(* Logix 5000 project; controller CLASE_1 Emulate 5570 rev 28.11; software revision 28.02; part 5 of 15 *)
(* tags used below, declared in another part *)
   P_Intlk : BOOL;   // Unique Parameter Name for auto - discovery
(* P_Intlk, continued *)

ROUTINE Prescan   (* ladder *)
// Clear "lurking" Commands
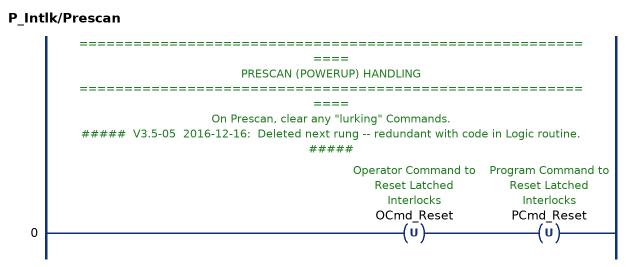
   // ============================================================
   // PRESCAN (POWERUP) HANDLING
   // ============================================================
   // On Prescan, clear any "lurking" Commands.
   // #####  V3.5-05  2016-12-16:  Deleted next rung -- redundant with code in Logic routine.  #####
   0: OTU(OCmd_Reset)OTU(PCmd_Reset);
END_ROUTINE
END_ADD_ON_INSTRUCTION

ADD_ON_INSTRUCTION P_Mode   (* revision 3.5 01 Release, vendor Rockwell Automation, ExecutePrescan, ExecuteEnableInFalse *)
// Mode
// Revision note:
// See V3.5-xx Release Notes for details. Unmodified, up-rev only for V3.5-01 Release.
// Help:
// Copyright © Rockwell Automation, Inc.  All Rights Reserved.
// This instruction provides selection of Mode (owner) for a Device level
// object  (from highest priority to lowest):
// *  No Mode (no owner, EnableIn is false)
// *  Hand (typically tracks hardwired control of device)
// *  Maint (Maintenance) (taken out of normal service for maintenance)
// *  Ovrd (Override) (typically used for process overrides)
// *  Prog  (Program) (automated control, and default if Cfg_ProgNorm = 1)
// *  Oper (Operator (manual control, and default if Cfg_ProgNorm = 0)
// (Program and Operator have the same priority.)
// The current mode is shown with Status bits and also as the primary
// Value for the instruction: an enumeration "Val" as follows:
//   0 = No Mode,
//   1 = Hand,
//   2 = Maintenance,
//   3 = Override,
//   4 = Program (Locked),
//   5 = Operator (Locked),
//   6 = Program (Unlocked, Oper default),
//   7 = Operator (Unlocked, Prog default),
//   8 = Program (Unlocked, = default),
//   9 = Operator (Unlocked, = default).
// When EnableIn is false, all ownership acquire/release and lock/unlock
// Commands are processed "behind the scenes", but the Mode is shown
// as "No Mode" (no owner).  When EnableIn becomes true, the Mode
// takes into account the Commands received -- in other words, the Mode
// becomes the one that would have been in effect had the EnableIn
// False / No Mode condition never occurred.
VAR_INPUT
   Inp_Hand : BOOL; {visible}   // 1=Acquire Hand (typ. hardwired local) Mode, 0=Release Hand Mode
   Inp_Ovrd : BOOL; {visible}   // 1=Acquire Override (higher priority program logic) Mode, 0=Release Override Mode
   Cfg_PCmdClear : BOOL := 1;   // 1=Clear Program Command on receipt; 0=Use Level-based (maintained) PCmds
   Cfg_OvrdOverLock : BOOL := 1;   // 1=Override supersedes Prog/Oper Lock, 0=don't override Lock
   Cfg_ProgDefault : BOOL;   // Default Mode: 1=Program Mode if no requests; 0=Operator Mode if no requests
   PCmd_Acq : BOOL;   // Program Command to Acquire Ownership (Oper to Prog)
   PCmd_Rel : BOOL;   // Program Command to Release Ownership (Prog to Oper)
   PCmd_Lock : BOOL;   // Program Command to Lock Mode in Prog
   PCmd_Unlock : BOOL;   // Program Command to Unlock Mode
   MCmd_Acq : BOOL;   // Maintenance Command to Acquire Ownership (Oper/Prog/Ovrd to Maint)
   MCmd_Rel : BOOL;   // Maintenance Command to Release Ownership (Maint to Oper/Prog/Ovrd)
   OCmd_AcqLock : BOOL;   // Operator Command to Acquire (Prog to Oper) / Lock Ownership
   OCmd_UnlockRel : BOOL;   // Operator Command to Unlock / Release (Oper to Prog) Ownership
END_VAR
VAR_OUTPUT
   Val : SINT; {access Read Only}   // Mode enum: 0=No, 1=H, 2=M, 3=!, 4=P Lock, 5=O Lock, 6=P (O Def), 7=O (P Def), 8=P (= Def), 9=O (= Def)
   Sts_Hand : BOOL; {access Read Only, visible}   // 1=Mode is Hand (supersedes Maint, Ovrd, Prog, Oper)
   Sts_Maint : BOOL; {access Read Only, visible}   // 1=Mode is Maintenance (supersedes Ovrd, Prog, Oper)
   Sts_Ovrd : BOOL; {access Read Only, visible}   // 1=Mode is Override (supersedes Prog, Oper)
   Sts_Prog : BOOL; {access Read Only, visible}   // 1=Mode is Program
   Sts_Oper : BOOL := 1; {access Read Only, visible}   // 1=Mode is Operator
   Sts_ProgOperLock : BOOL; {access Read Only, visible}   // 1=Program or Operator has requested Mode Lock
   Sts_ProgOperSel : BOOL; {access Read Only}   // Prog/Oper selection 1=Program, 0=Operator
   Sts_NoMode : BOOL; {access Read Only}   // 1=Mode is No Mode (no owner, disabled or not scanned)
   Sts_MAcqRcvd : BOOL; {access Read Only}   // 1=Maintenance Acquire command received this scan
   Rdy_MAcq : BOOL; {access Read Only}   // 1=Ready for MCmd_Acq, enable button
   Rdy_MRel : BOOL; {access Read Only}   // 1=Ready for MCmd_Rel, enable button
   Rdy_OAcq : BOOL; {access Read Only}   // 1=Ready for OCmd_AcqLock, enable Acquire (to Oper) button
   Rdy_OLock : BOOL; {access Read Only}   // 1=Ready for OCmd_AcqLock, enable Oper Lock button
   Rdy_OUnlock : BOOL; {access Read Only}   // 1=Ready for OCmd_UnlockRel, enable Oper Unlock button
   Rdy_ORel : BOOL; {access Read Only}   // 1=Ready for OCmd_UnlockRel, enable Release (to Prog) button
   P_Mode : BOOL;   // Unique Parameter Name for auto - discovery
END_VAR
VAR
   Wrk_Locked : BOOL; {access None}   // 1=Program/Operator Mode selection is Locked
   Wrk_Prog : BOOL; {access None}   // Internal Program (1) / Operator (0) Mode selection
   Wrk_Maint : BOOL; {access None}   // Internal Maintenance Mode
   Inf_Lib : STRING_12 := 'RA-BAS'; {access Read Only}   // Display Library for Faceplate call-up
   Inf_Type : STRING_16 := 'P_Mode'; {access Read Only}   // Must contain AOI name, used for HMI and Information S/W
END_VAR

ROUTINE EnableInFalse   (* ladder *)
// Processes received Commands, but shows "NO mode" (no owner)
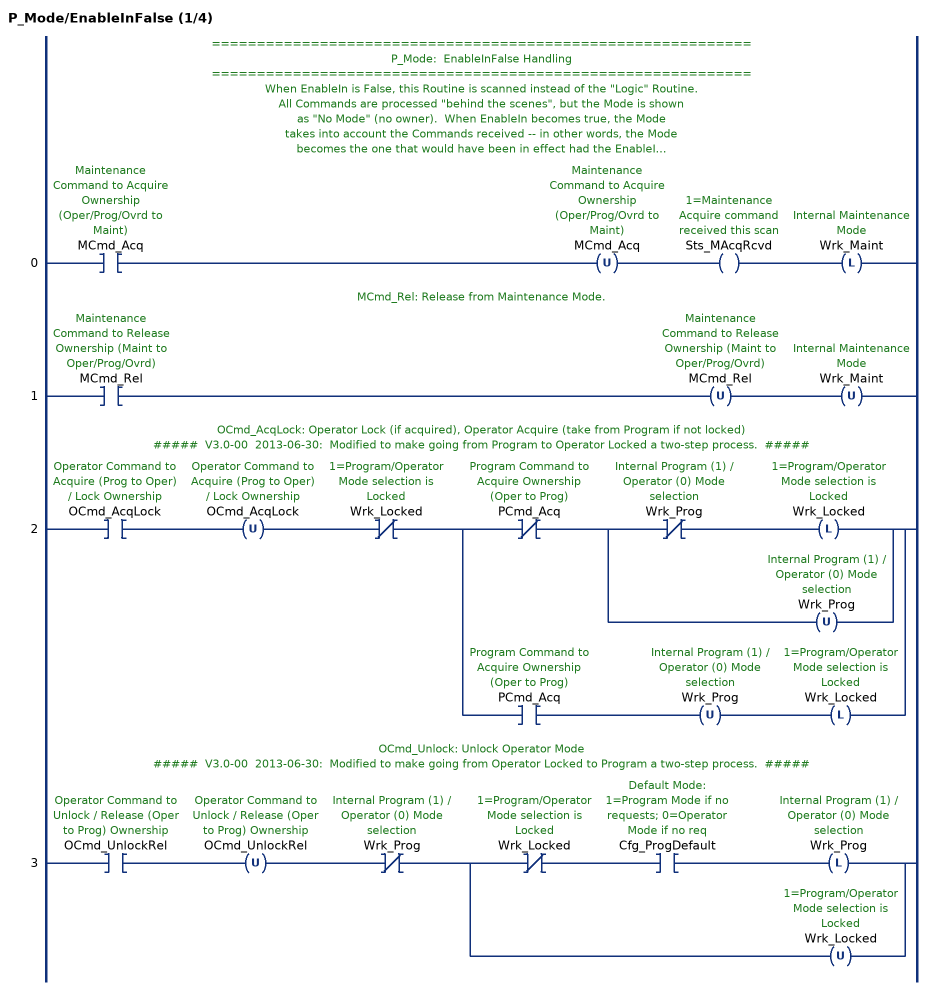
   // ============================================================
   // P_Mode:  EnableInFalse Handling
   // ============================================================
   // When EnableIn is False, this Routine is scanned instead of the "Logic" Routine.
   // All Commands are processed "behind the scenes", but the Mode is shown
   // as "No Mode" (no owner).  When EnableIn becomes true, the Mode
   // takes into account the Commands received -- in other words, the Mode
   // becomes the one that would have been in effect had the EnableIn
   // False / No Mode condition never occurred.
   // ============================================================
   // COMMAND HANDLING
   // ============================================================
   // NOTE:  These rungs MUST be in the order given to meet the following
   // multiple-actions-at-the-same-time scenarios:
   // * Maintenance Release beats Maintenance Acquire
   // * Program Release beats Program Acquire
   // * Program Unlock beats Program Lock
   // * Operator Unlock beats Operator Acquire and Lock (results in Oper Unlocked)
   // * Operator Acquire/Lock must come after Program Unlock
   // * Program Acquire must come after Operator Unlock
   // ===========================================================
   // MCmd_Acq: Acquire for Maintenance Mode, and blink the status
   // that indicates a Maintenance Acquire command was received.
   // #####  V3.1-00  2014-06-30:  Added Sts_MAcqRcvd  #####
   0: XIC(MCmd_Acq)OTU(MCmd_Acq)OTE(Sts_MAcqRcvd)OTL(Wrk_Maint);
   // MCmd_Rel: Release from Maintenance Mode.
   1: XIC(MCmd_Rel)OTU(MCmd_Rel)OTU(Wrk_Maint);
   // OCmd_AcqLock: Operator Lock (if acquired), Operator Acquire (take from Program if not locked)
   // #####  V3.0-00  2013-06-30:  Modified to make going from Program to Operator Locked a two-step process.  #####
   2: XIC(OCmd_AcqLock)OTU(OCmd_AcqLock)XIO(Wrk_Locked)[XIO(PCmd_Acq) [XIO(Wrk_Prog) OTL(Wrk_Locked) ,OTU(Wrk_Prog) ] ,XIC(PCmd_Acq) OTU(Wrk_Prog) OTL(Wrk_Locked) ];
   // OCmd_Unlock: Unlock Operator Mode
   // #####  V3.0-00  2013-06-30:  Modified to make going from Operator Locked to Program a two-step process.  #####
   3: XIC(OCmd_UnlockRel)OTU(OCmd_UnlockRel)XIO(Wrk_Prog)[XIO(Wrk_Locked) XIC(Cfg_ProgDefault) OTL(Wrk_Prog) ,OTU(Wrk_Locked) ];
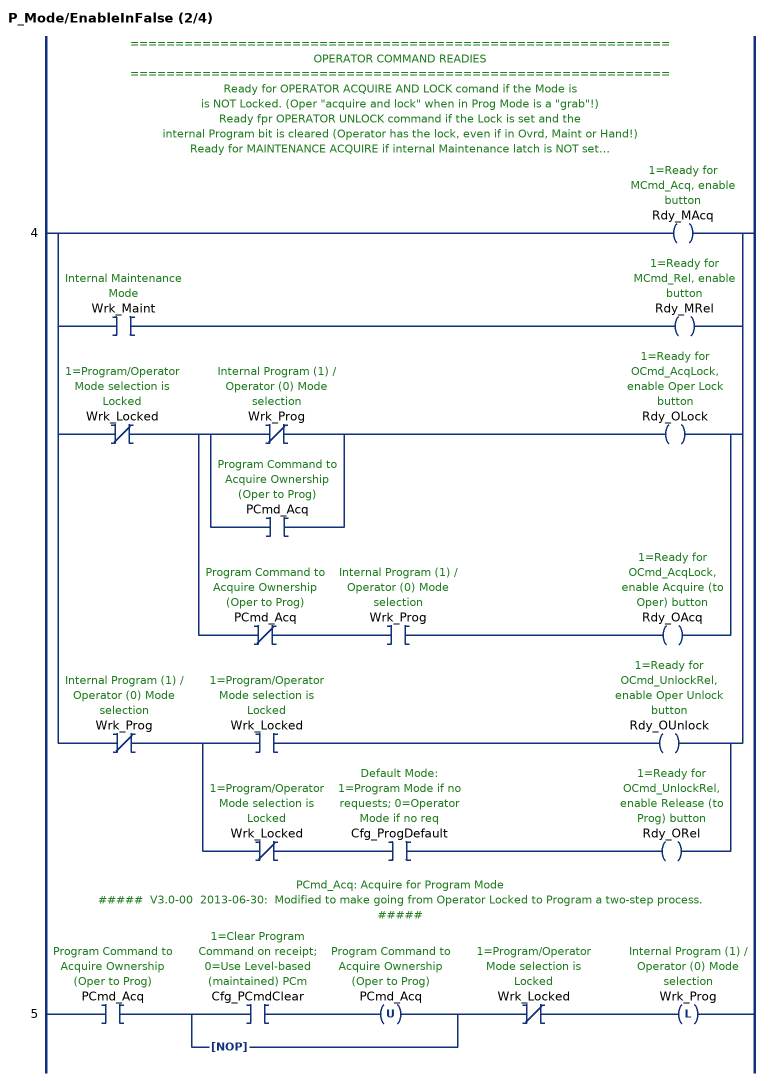
   // ============================================================
   // OPERATOR COMMAND READIES
   // ============================================================
   // Ready for OPERATOR ACQUIRE AND LOCK comand if the Mode is
   //  is NOT Locked. (Oper "acquire and lock" when in Prog Mode is a "grab"!)
   // Ready fpr OPERATOR UNLOCK command if the Lock is set and the
   // internal Program bit is cleared (Operator has the lock, even if in Ovrd, Maint or Hand!)
   // Ready for MAINTENANCE ACQUIRE if internal Maintenance latch is NOT set.
   // But we need to display Ready even if latch IS set so that Sts_MAcqRcvd
   // can blink to reset an external Maintenance expiration timer!!!
   // Ready for MAINTENANCE RELEASE if internal Maintenance latch IS set.
   // #####  V3.0-00  2013-06-30:  Modified Rdy_Unlock for two-step Operator Locked to Program process.  #####
   // #####  V3.1-00  2014-06-30:  Added Sts_MAcqRcvd  #####
   4: [OTE(Rdy_MAcq) ,XIC(Wrk_Maint) OTE(Rdy_MRel) ,XIO(Wrk_Locked) [[XIO(Wrk_Prog) ,XIC(PCmd_Acq) ] OTE(Rdy_OLock) ,XIO(PCmd_Acq) XIC(Wrk_Prog) OTE(Rdy_OAcq) ] ,XIO(Wrk_Prog) [XIC(Wrk_Locked) OTE(Rdy_OUnlock) ,XIO(Wrk_Locked) XIC(Cfg_ProgDefault) OTE(Rdy_ORel) ] ];
   // PCmd_Acq: Acquire for Program Mode
   // #####  V3.0-00  2013-06-30:  Modified to make going from Operator Locked to Program a two-step process.  #####
   5: XIC(PCmd_Acq)[XIC(Cfg_PCmdClear) OTU(PCmd_Acq) ,NOP() ]XIO(Wrk_Locked)OTL(Wrk_Prog);
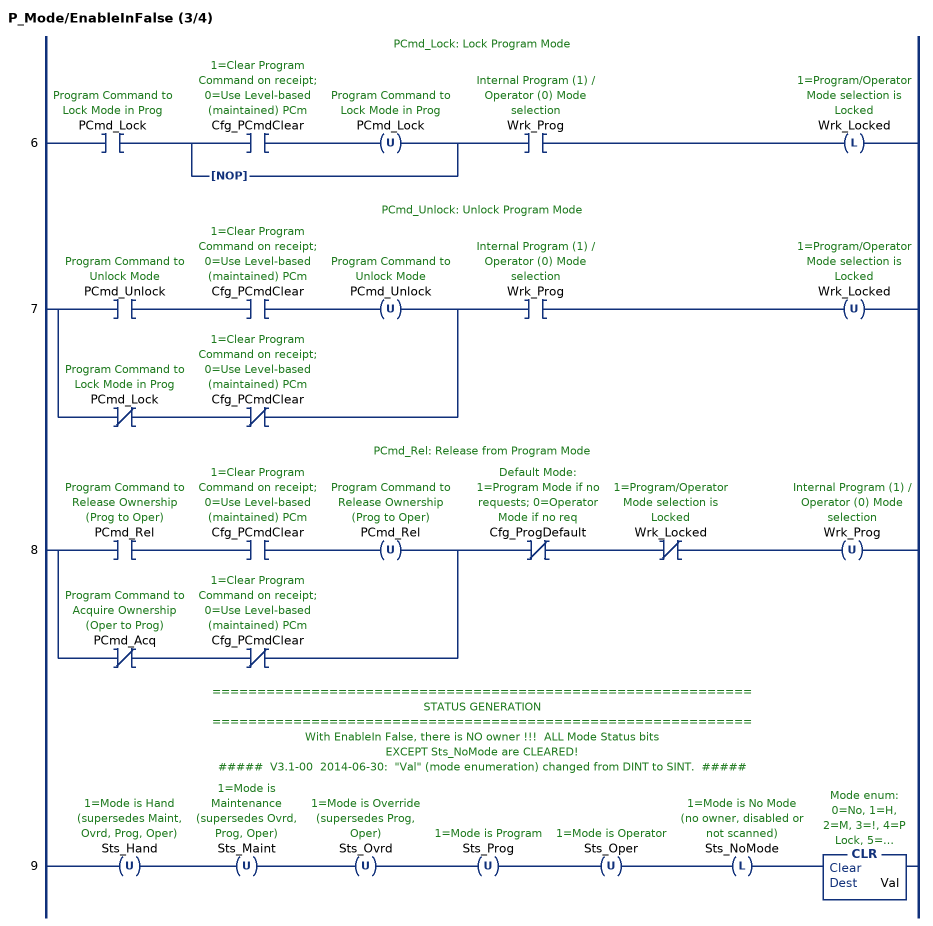
   // PCmd_Lock: Lock Program Mode
   6: XIC(PCmd_Lock)[XIC(Cfg_PCmdClear) OTU(PCmd_Lock) ,NOP() ]XIC(Wrk_Prog)OTL(Wrk_Locked);
   // PCmd_Unlock: Unlock Program Mode
   7: [XIC(PCmd_Unlock) XIC(Cfg_PCmdClear) OTU(PCmd_Unlock) ,XIO(PCmd_Lock) XIO(Cfg_PCmdClear) ]XIC(Wrk_Prog)OTU(Wrk_Locked);
   // PCmd_Rel: Release from Program Mode
   8: [XIC(PCmd_Rel) XIC(Cfg_PCmdClear) OTU(PCmd_Rel) ,XIO(PCmd_Acq) XIO(Cfg_PCmdClear) ]XIO(Cfg_ProgDefault)XIO(Wrk_Locked)OTU(Wrk_Prog);
   // ============================================================
   // STATUS GENERATION
   // ============================================================
   // With EnableIn False, there is NO owner !!!  ALL Mode Status bits
   // EXCEPT Sts_NoMode are CLEARED!
   // #####  V3.1-00  2014-06-30:  "Val" (mode enumeration) changed from DINT to SINT.  #####
   9: OTU(Sts_Hand)OTU(Sts_Maint)OTU(Sts_Ovrd)OTU(Sts_Prog)OTU(Sts_Oper)OTL(Sts_NoMode)CLR(Val);
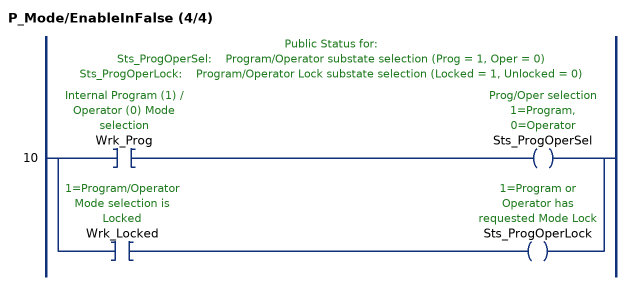
   // Public Status for:
   // Sts_ProgOperSel:    Program/Operator substate selection (Prog = 1, Oper = 0)
   // Sts_ProgOperLock:    Program/Operator Lock substate selection (Locked = 1, Unlocked = 0)
   10: [XIC(Wrk_Prog) OTE(Sts_ProgOperSel) ,XIC(Wrk_Locked) OTE(Sts_ProgOperLock) ];
END_ROUTINE

ROUTINE Logic   (* ladder *)
// Selects Modes (Hand, Maint, Ovrd, Oper, Prog) based on Inputs and Commands
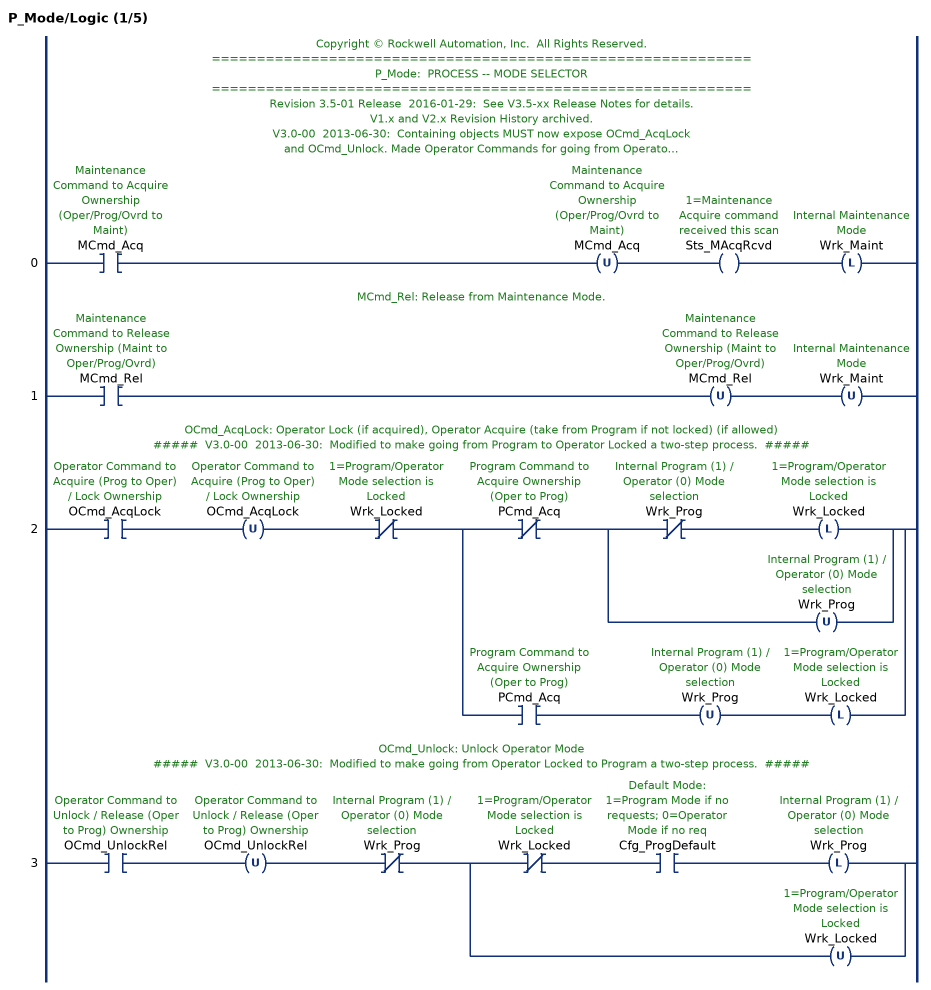
   // Copyright © Rockwell Automation, Inc.  All Rights Reserved.
   // ============================================================
   // P_Mode:  PROCESS -- MODE SELECTOR
   // ============================================================
   // Revision 3.5-01 Release  2016-01-29:  See V3.5-xx Release Notes for details.
   // V1.x and V2.x Revision History archived.
   // V3.0-00  2013-06-30:  Containing objects MUST now expose OCmd_AcqLock
   // and OCmd_Unlock. Made Operator Commands for going from Operator
   // Locked to Program (unlocked) and Program (unlocked) to Operator
   // Lock two-step processes.  Added Inf_Lib, Inf_Type.
   // V3.1-00  2014-06-30:  Containing objects must expose Maintenance Acquire /
   // Release commands and new Sts_MAcqRcvd.
   // Changed Val (enum) to SINT. Fixed parameter descriptions.
   // V3.1-01  2014-09-03:  Unmodified, up-rev only for V3.1-01 public release.
   // V3.5-01  2016-01-29:  Unmodified, up-rev only for V3.5-01 Release.
   // ============================================================
   // This instruction provides selection of Mode (owner) for a Device level
   // object  (from highest priority to lowest):
   // * NO Mode (EnableIn is false)
   // *  Hand (typically tracks hardwired control of device)
   // *  Maint (Maintenance) (taken out of normal service for maintenance)
   // *  Ovrd (Override) (typically used for process overrides)
   // *  Prog  (Program) (automated control, and default if Cfg_ProgNorm = 1)
   // *  Oper (Operator (manual control, and default if Cfg_ProgNorm = 0)
   // The current mode is shown with Status bits and also as the
   // primary Value for the instruction: an enumeration as follows:
   // 0 = No Mode, 1 = Hand, 2 = Maintenance, 3 = Override,
   // 4 = Program (Locked), 5 = Operator (Locked),
   // 6 = Program (Unlocked, Oper default), 7 = Operator (Unlocked, Prog default),
   // 8 = Program (Unlocked, Prog default), 9 = Operator (Unlocked, Oper default).
   // ============================================================
   // COMMAND HANDLING
   // ============================================================
   // NOTE:  These rungs MUST be in the order given to meet the following
   // multiple-actions-at-the-same-time scenarios:
   // * Maintenance Release beats Maintenance Acquire
   // * Program Release beats Program Acquire
   // * Program Unlock beats Program Lock
   // * Operator Unlock beats Operator Acquire / Lock (results in Oper Unlocked)
   // * Program Acquire must come after Operator Unlock
   // If Cfg_ProgDefault = 1, the Mode defaults to Program
   // (instead of Operator) if all other Modes release their requests.
   // ============================================================
   // MCmd_Acq: Acquire for Maintenance Mode, and blink the status
   // that indicates a Maintenance Acquire command was received.
   // #####  V3.1-00  2014-06-30:  Added Sts_MAcqRcvd  #####
   0: XIC(MCmd_Acq)OTU(MCmd_Acq)OTE(Sts_MAcqRcvd)OTL(Wrk_Maint);
   // MCmd_Rel: Release from Maintenance Mode.
   1: XIC(MCmd_Rel)OTU(MCmd_Rel)OTU(Wrk_Maint);
   // OCmd_AcqLock: Operator Lock (if acquired), Operator Acquire (take from Program if not locked) (if allowed)
   // #####  V3.0-00  2013-06-30:  Modified to make going from Program to Operator Locked a two-step process.  #####
   2: XIC(OCmd_AcqLock)OTU(OCmd_AcqLock)XIO(Wrk_Locked)[XIO(PCmd_Acq) [XIO(Wrk_Prog) OTL(Wrk_Locked) ,OTU(Wrk_Prog) ] ,XIC(PCmd_Acq) OTU(Wrk_Prog) OTL(Wrk_Locked) ];
   // OCmd_Unlock: Unlock Operator Mode
   // #####  V3.0-00  2013-06-30:  Modified to make going from Operator Locked to Program a two-step process.  #####
   3: XIC(OCmd_UnlockRel)OTU(OCmd_UnlockRel)XIO(Wrk_Prog)[XIO(Wrk_Locked) XIC(Cfg_ProgDefault) OTL(Wrk_Prog) ,OTU(Wrk_Locked) ];
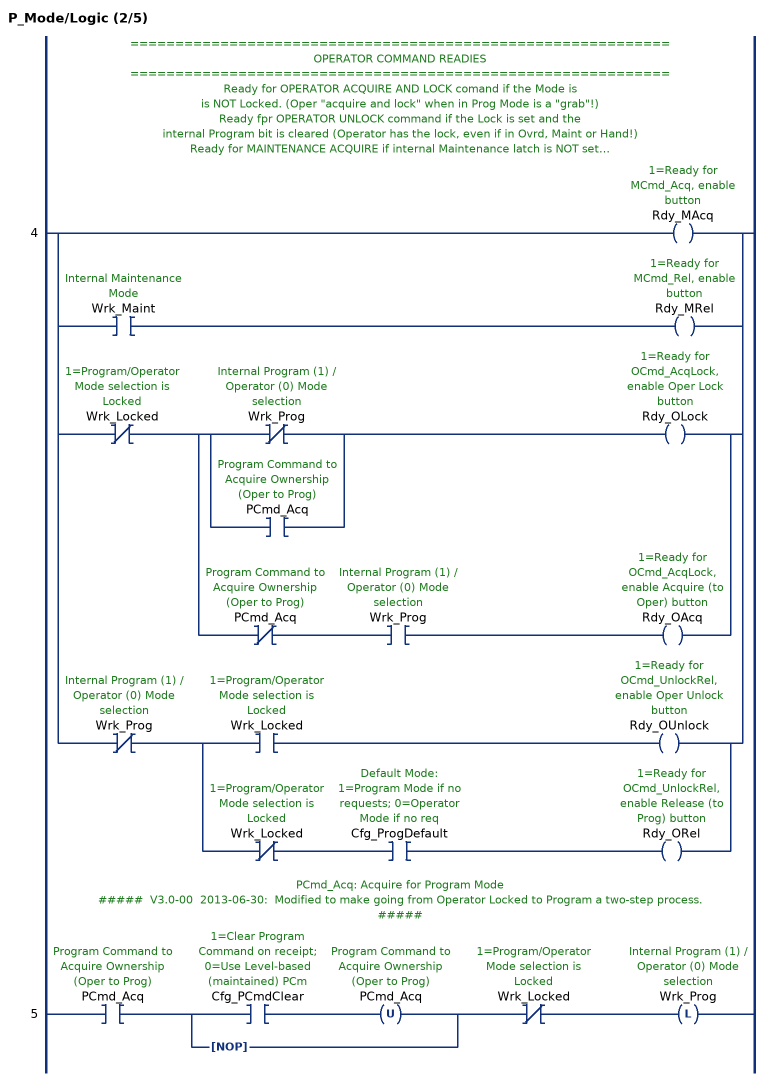
   // ============================================================
   // OPERATOR COMMAND READIES
   // ============================================================
   // Ready for OPERATOR ACQUIRE AND LOCK comand if the Mode is
   //  is NOT Locked. (Oper "acquire and lock" when in Prog Mode is a "grab"!)
   // Ready fpr OPERATOR UNLOCK command if the Lock is set and the
   // internal Program bit is cleared (Operator has the lock, even if in Ovrd, Maint or Hand!)
   // Ready for MAINTENANCE ACQUIRE if internal Maintenance latch is NOT set.
   // But we need to display Ready even if latch IS set so that Sts_MAcqRcvd
   // can blink to reset an external Maintenance expiration timer!!!
   // Ready for MAINTENANCE RELEASE if internal Maintenance latch IS set.
   // #####  V3.0-00  2013-06-30:  Modified Rdy_Unlock for two-step Operator Locked to Program process.  #####
   // #####  V3.1-00  2014-06-30:  Added Sts_MAcqRcvd  #####
   4: [OTE(Rdy_MAcq) ,XIC(Wrk_Maint) OTE(Rdy_MRel) ,XIO(Wrk_Locked) [[XIO(Wrk_Prog) ,XIC(PCmd_Acq) ] OTE(Rdy_OLock) ,XIO(PCmd_Acq) XIC(Wrk_Prog) OTE(Rdy_OAcq) ] ,XIO(Wrk_Prog) [XIC(Wrk_Locked) OTE(Rdy_OUnlock) ,XIO(Wrk_Locked) XIC(Cfg_ProgDefault) OTE(Rdy_ORel) ] ];
   // PCmd_Acq: Acquire for Program Mode
   // #####  V3.0-00  2013-06-30:  Modified to make going from Operator Locked to Program a two-step process.  #####
   5: XIC(PCmd_Acq)[XIC(Cfg_PCmdClear) OTU(PCmd_Acq) ,NOP() ]XIO(Wrk_Locked)OTL(Wrk_Prog);
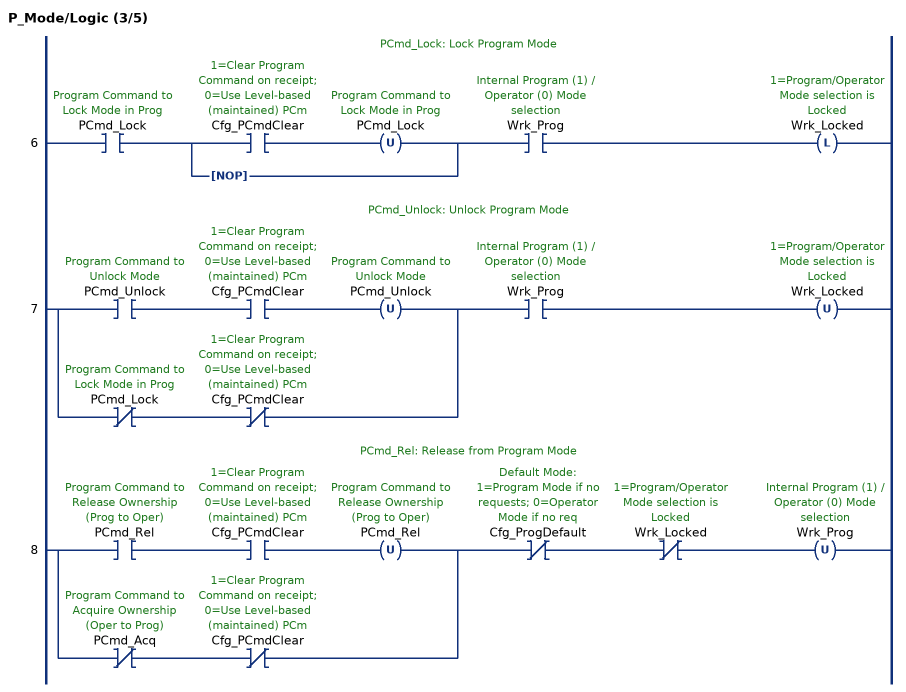
   // PCmd_Lock: Lock Program Mode
   6: XIC(PCmd_Lock)[XIC(Cfg_PCmdClear) OTU(PCmd_Lock) ,NOP() ]XIC(Wrk_Prog)OTL(Wrk_Locked);
   // PCmd_Unlock: Unlock Program Mode
   7: [XIC(PCmd_Unlock) XIC(Cfg_PCmdClear) OTU(PCmd_Unlock) ,XIO(PCmd_Lock) XIO(Cfg_PCmdClear) ]XIC(Wrk_Prog)OTU(Wrk_Locked);
   // PCmd_Rel: Release from Program Mode
   8: [XIC(PCmd_Rel) XIC(Cfg_PCmdClear) OTU(PCmd_Rel) ,XIO(PCmd_Acq) XIO(Cfg_PCmdClear) ]XIO(Cfg_ProgDefault)XIO(Wrk_Locked)OTU(Wrk_Prog);
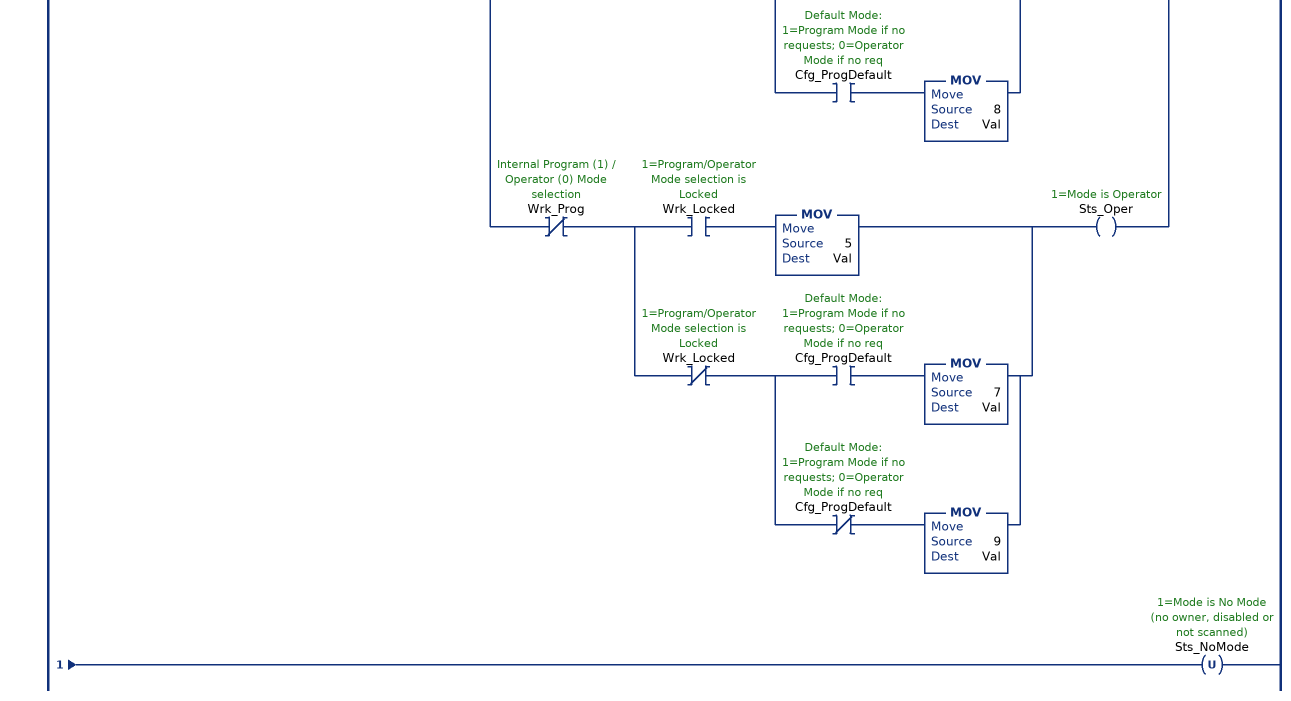
   // ============================================================
   // STATUS GENERATION
   // ============================================================
   // This rung determines the Mode based on the states of the inputs and internal working bits.
   // The logic here does the vast mahority of the implementation of the Mode selection rules.
   // Between the internal working bits used above and the rules implemented here,
   // outside objects cannot manipulate the state of this object by setting/clearing its Status bits.
   // Public Status is generated for:
   // *  Hand Mode
   // *  Maintenance Mode
   // *  Override Mode
   // *  Program Mode
   // *  Operator Mode
   // *  No Mode (none of the above)
   // #####  V3.1-00  2014-06-30:  "Val" (mode enumeration) changed from DINT to SINT.  #####
   9: [XIC(Inp_Hand) OTE(Sts_Hand) MOV(1,Val) ,XIO(Inp_Hand) [XIC(Wrk_Maint) OTE(Sts_Maint) MOV(2,Val) ,XIO(Wrk_Maint) [XIC(Inp_Ovrd) [XIO(Wrk_Locked) ,XIC(Cfg_OvrdOverLock) ,XIC(Sts_Ovrd) ] OTE(Sts_Ovrd) MOV(3,Val) ,XIO(Sts_Ovrd) [XIC(Wrk_Prog) [XIC(Wrk_Locked) MOV(4,Val) ,XIO(Wrk_Locked) [XIO(Cfg_ProgDefault) MOV(6,Val) ,XIC(Cfg_ProgDefault) MOV(8,Val) ] ] OTE(Sts_Prog) ,XIO(Wrk_Prog) [XIC(Wrk_Locked) MOV(5,Val) ,XIO(Wrk_Locked) [XIC(Cfg_ProgDefault) MOV(7,Val) ,XIO(Cfg_ProgDefault) MOV(9,Val) ] ] OTE(Sts_Oper) ] ] ] ]OTU(Sts_NoMode);
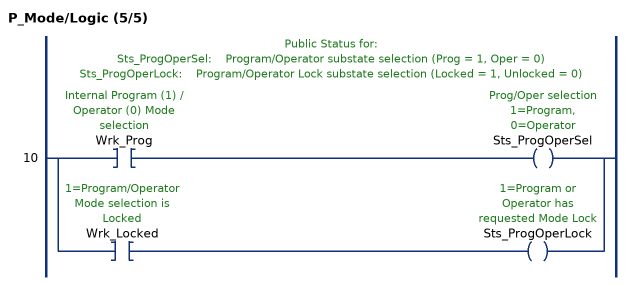
   // Public Status for:
   // Sts_ProgOperSel:    Program/Operator substate selection (Prog = 1, Oper = 0)
   // Sts_ProgOperLock:    Program/Operator Lock substate selection (Locked = 1, Unlocked = 0)
   10: [XIC(Wrk_Prog) OTE(Sts_ProgOperSel) ,XIC(Wrk_Locked) OTE(Sts_ProgOperLock) ];
END_ROUTINE

ROUTINE Prescan   (* ladder *)
// Clear "lurking" Commands
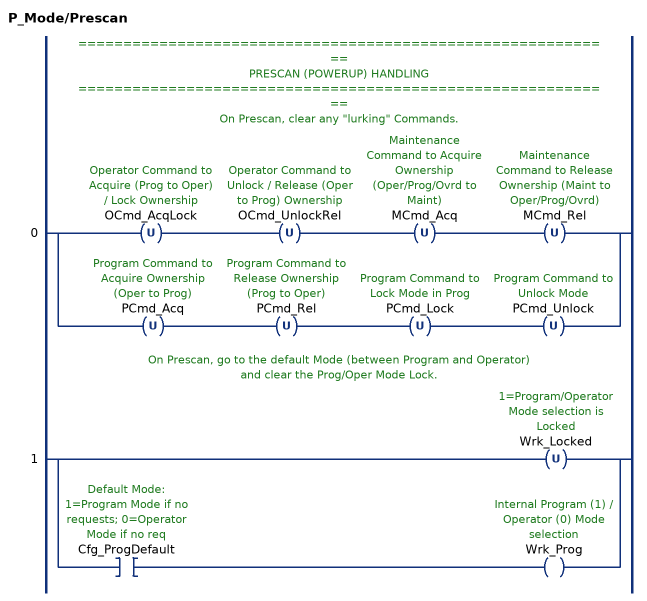
   // ============================================================
   // PRESCAN (POWERUP) HANDLING
   // ============================================================
   // On Prescan, clear any "lurking" Commands.
   0: [OTU(OCmd_AcqLock) OTU(OCmd_UnlockRel) OTU(MCmd_Acq) OTU(MCmd_Rel) ,OTU(PCmd_Acq) OTU(PCmd_Rel) OTU(PCmd_Lock) OTU(PCmd_Unlock) ];
   // On Prescan, go to the default Mode (between Program and Operator)
   // and clear the Prog/Oper Mode Lock.
   1: [OTU(Wrk_Locked) ,XIC(Cfg_ProgDefault) OTE(Wrk_Prog) ];
END_ROUTINE
END_ADD_ON_INSTRUCTION

ADD_ON_INSTRUCTION P_Motor   (* revision 3.5 09 Release, vendor Rockwell Automation, ExecutePrescan, ExecuteEnableInFalse *)
// Single Speed Motor
// Revision note:
// See V3.5-xx Release Notes for details. Modified to correct indication of motor RUNNING status in HAND mode, regardless of interlock/stop conditions.
// Help:
// Copyright © Rockwell Automation, Inc.  All Rights Reserved.
// This Instruction controls and monitors a single-speed motor
// (FVNR, soft-start, etc.) and provides:
// *  Monitoring of run feedback, display of actual motor status
// *  Detection of Failure to Start, Failure to Stop
// *  Monitoring of a Permissive condition to allow starting
// *  Monitoring of an Interlock condition to stop / prevent starting
// *  Simulation, providing feedback of a working motor while disabling outputs
// *  Monitoring of I/O communication faults
// *  Alarms for Fail to Start, Fail to Stop, Interlock Trip, I/O Fault
// *  Options to shed (stop motor) on Fail to Start or I/O Fault
// *  Operation in Hand, Maintenance, Override, Program and Operator Modes
// *  Option to automatically reset faults and alarms when operator commands
//      motor to start or stop
// *  Supports HMI "breadcrumbs" for Alarm Inhibited, Bad Configuration,
//      Not Ready, Maintenance Bypass Active
// *  "Available" status for use by automation logic to know whether motor
//      can be controlled by other objects.
// Modes are provided by a P_Mode AOI instance.
// Alarms are provided by P_Alarm AOI instances.
// Modes of operation: Operator, Program, Override, Maintenance, Hand
VAR_INPUT
   Inp_RunFdbk : BOOL; {visible}   // Input Signal: RUN feedback from motor
   Inp_PermOK : BOOL := 1; {visible}   // 1=Permissives OK, motor can start
   Inp_NBPermOK : BOOL := 1; {visible}   // 1=Non-Bypassable Permissives OK, motor can start
   Inp_IntlkOK : BOOL := 1; {visible}   // 1=Interlocks OK, motor can start/run
   Inp_NBIntlkOK : BOOL := 1; {visible}   // 1=Non-Bypassable Interlocks OK, motor can start/run
   Inp_IOFault : BOOL;   // Input Communication Status 0=OK, 1=fail
   Inp_Sim : BOOL;   // 1=Simulate working motor; 0=Start/Stop/ Monitor actual motor
   Inp_Hand : ALIAS FOR Mode.Inp_Hand;
   Inp_Ovrd : ALIAS FOR Mode.Inp_Ovrd;
   Inp_OvrdCmd : DINT;   // Override Mode Command: 0=None, 1=Stop, 2=Start
   Inp_Reset : BOOL;   // 1=Reset all fault conditions and latched Alarms
   Cfg_HasRunFdbk : BOOL;   // 1=Motor provides run feedback
   Cfg_UseRunFdbk : BOOL;   // 1=Motor run feedback should be used for failure checking
   Cfg_AllowLocal : BOOL;   // 1=Allow Local Start/Stop without alarm, 0=Start/Stop from HMI/prog only
   Cfg_HasPermObj : BOOL;   // 1=Enable navigation to permissive object
   Cfg_HasIntlkObj : BOOL;   // 1=Enable navigation to interlock object
   Cfg_HasResInhObj : BOOL;   // 1=Enable navigation to restart inhibit object
   Cfg_HasRunTimeObj : BOOL;   // 1=Enable navigation to run time object
   Cfg_HasOvldObj : BOOL;   // 1=Enable navigation to overload object
   Cfg_PCmdClear : ALIAS FOR Mode.Cfg_PCmdClear;
   Cfg_ProgDefault : ALIAS FOR Mode.Cfg_ProgDefault;
   Cfg_OperStopPrio : BOOL;   // 1=OCmd_Stop available in any mode, 0=OCmd_Stop only in Oper, Maint modes.
   Cfg_OCmdResets : BOOL;   // 1=New Oper motor cmd. resets fault, 0=reset req'd to clear fault
   Cfg_OvrdPermIntlk : BOOL;   // 1=Override ignores Bypassable Perm/ Intlk; 0=always use Perm/Intlk
   Cfg_ShedOnFailToStart : BOOL := 1;   // 1=Stop Motor and Alarm on Fail to Start; 0=Alarm only on Fail to Start
   Cfg_ShedOnIOFault : BOOL := 1;   // 1=Stop Motor and Alarm on I/O Fault; 0=Alarm only on I/O Fault
   Cfg_HasFailToStartAlm : ALIAS FOR FailToStart.Cfg_Exists;   // 1=Fail to Start Alarm exists and will be checked
   Cfg_HasFailToStopAlm : ALIAS FOR FailToStop.Cfg_Exists;   // 1=Fail to Stop Alarm exists and will be checked
   Cfg_HasIntlkTripAlm : ALIAS FOR IntlkTrip.Cfg_Exists;   // 1=Interlock Trip Alarm exists and will be checked
   Cfg_HasIOFaultAlm : ALIAS FOR IOFault.Cfg_Exists;   // 1=I/O Fault Alarm exists and will be checked
   Cfg_FailToStartResetReqd : ALIAS FOR FailToStart.Cfg_ResetReqd;   // 1=Reset required to clear Fail to Start Alarm
   Cfg_FailToStopResetReqd : ALIAS FOR FailToStop.Cfg_ResetReqd;   // 1=Reset required to clear Fail to Stop Alarm
   Cfg_IntlkTripResetReqd : ALIAS FOR IntlkTrip.Cfg_ResetReqd;   // 1=Reset required to clear Interlock Trip Alarm
   Cfg_IOFaultResetReqd : ALIAS FOR IOFault.Cfg_ResetReqd;   // 1=Reset required to clear I/O Fault Alarm
   Cfg_FailToStartAckReqd : ALIAS FOR FailToStart.Cfg_AckReqd;   // 1=Acknowledge required for Fail to Start Alarm
   Cfg_FailToStopAckReqd : ALIAS FOR FailToStop.Cfg_AckReqd;   // 1=Acknowledge required for Fail to Stop Alarm
   Cfg_IntlkTripAckReqd : ALIAS FOR IntlkTrip.Cfg_AckReqd;   // 1=Acknowledge required for Interlock Trip Alarm
   Cfg_IOFaultAckReqd : ALIAS FOR IOFault.Cfg_AckReqd;   // 1=Acknowledge required for I/O Fault Alarm
   Cfg_FailToStartSeverity : ALIAS FOR FailToStart.Cfg_Severity;   // Fail To Start Alarm Severity: 1..250=Low, 251..500=Medium, 501..750=High, 751..1000=Urgent
   Cfg_FailToStopSeverity : ALIAS FOR FailToStop.Cfg_Severity;   // Fail To Stop Alarm Severity: 1..250=Low, 251..500=Medium, 501..750=High, 751..1000=Urgent
   Cfg_IntlkTripSeverity : ALIAS FOR IntlkTrip.Cfg_Severity;   // Interlock Trip Alarm Severity: 1..250=Low, 251..500=Medium, 501..750=High, 751..1000=Urgent
   Cfg_IOFaultSeverity : ALIAS FOR IOFault.Cfg_Severity;   // I/O Fault Alarm Severity: 1..250=Low, 251..500=Medium, 501..750=High, 751..1000=Urgent
   Cfg_SimFdbkT : DINT := 2;   // Feedback delay in Simulation (sec)
   Cfg_FailToStartT : DINT := 10;   // Time after Start for running feedback before Fault (sec)
   Cfg_FailToStopT : DINT := 10;   // Time after Stop for stopped feedback (=0) before Fault (sec)
   PSet_Owner : DINT;   // Program Owner Request ID (non-zero) or Release (zero)
   PCmd_Start : BOOL;   // Program Command to Start Motor
   PCmd_Stop : BOOL;   // Program Command to Stop Motor
   PCmd_Acq : ALIAS FOR Mode.PCmd_Acq;
   PCmd_Rel : ALIAS FOR Mode.PCmd_Rel;
   PCmd_Lock : ALIAS FOR Mode.PCmd_Lock;
   PCmd_Unlock : ALIAS FOR Mode.PCmd_Unlock;
   PCmd_Reset : BOOL;   // Program Command to Reset all Alarms requiring Reset
   PCmd_FailToStartAck : ALIAS FOR FailToStart.PCmd_Ack;   // Program Command to Acknowledge Fail to Start Alarm
   PCmd_FailToStartSuppress : ALIAS FOR FailToStart.PCmd_Suppress;   // Program Command to Suppress Fail to Start Alarm
   PCmd_FailToStartUnsuppress : ALIAS FOR FailToStart.PCmd_Unsuppress;   // Program Command to Unsuppress Fail to Start Alarm
   PCmd_FailToStartUnshelve : ALIAS FOR FailToStart.PCmd_Unshelve;   // Program Command to Unshelve Fail to Start Alarm
   PCmd_FailToStopAck : ALIAS FOR FailToStop.PCmd_Ack;   // Program Command to Acknowledge Fail to Stop Alarm
   PCmd_FailToStopSuppress : ALIAS FOR FailToStop.PCmd_Suppress;   // Program Command to Suppress Fail to Stop Alarm
   PCmd_FailToStopUnsuppress : ALIAS FOR FailToStop.PCmd_Unsuppress;   // Program Command to Unsuppress Fail to Stop Alarm
   PCmd_FailToStopUnshelve : ALIAS FOR FailToStop.PCmd_Unshelve;   // Program Comnmand to Unshelve Fail to Stop Alarm
   PCmd_IntlkTripAck : ALIAS FOR IntlkTrip.PCmd_Ack;   // Program Command to Acknowledge Interlock Trip Alarm
   PCmd_IntlkTripSuppress : ALIAS FOR IntlkTrip.PCmd_Suppress;   // Program Command to Suppress Interlock Trip Alarm
   PCmd_IntlkTripUnsuppress : ALIAS FOR IntlkTrip.PCmd_Unsuppress;   // Program Command to Unsuppress Interlock Trip Alarm
   PCmd_IntlkTripUnshelve : ALIAS FOR IntlkTrip.PCmd_Unshelve;   // Program Command to Unshelve Interlock Trip Alarm
   PCmd_IOFaultAck : ALIAS FOR IOFault.PCmd_Ack;   // Program Command to Acknowledge I/O Fault Alarm
   PCmd_IOFaultSuppress : ALIAS FOR IOFault.PCmd_Suppress;   // Program Command to Suppress I/O Fault Alarm
   PCmd_IOFaultUnsuppress : ALIAS FOR IOFault.PCmd_Unsuppress;   // Program Command to Unsuppress I/O Fault Alarm
   PCmd_IOFaultUnshelve : ALIAS FOR IOFault.PCmd_Unshelve;   // Program Command to Unshelve I/O Fault Alarm
   OCmd_Start : BOOL;   // Operator Command to Start Motor
   OCmd_Stop : BOOL;   // Operator Command to Stop Motor
   OCmd_Bypass : BOOL;   // Operator Command to Bypass all Bypassable Interlocks and Permissives
   OCmd_Check : BOOL;   // Operator Command to Check (not bypass) all Interlocks and Permissives
   MCmd_Disable : BOOL;   // Maintenance Command to Disable Motor
   MCmd_Enable : BOOL;   // Maintenance Command to Enable (allow to run) Motor
   MCmd_Acq : ALIAS FOR Mode.MCmd_Acq;
   MCmd_Rel : ALIAS FOR Mode.MCmd_Rel;
   OCmd_AcqLock : ALIAS FOR Mode.OCmd_AcqLock;
   OCmd_Unlock : ALIAS FOR Mode.OCmd_UnlockRel;
   OCmd_Reset : BOOL;   // Operator Command to Reset all Alarms requiring Reset
   OCmd_ResetAckAll : BOOL;   // Operator Command to Reset all Alarms and latched Shed conditions
END_VAR
VAR_OUTPUT
   Out_Run : BOOL; {access Read Only, visible}   // 1=Run Motor, 0=Stop Motor
   Out_Start : BOOL; {access Read Only, visible}   // 1=Start Motor, 0=Motor left in current state
   Out_Stop : BOOL; {access Read Only, visible}   // 1=Stop Motor, 0=Motor left in current state
   SrcQ_IO : SINT; {access Read Only}   // Source and Quality of primary I/O (enumeration)
   SrcQ : SINT; {access Read Only}   // Source and Quality of primary Val/Sts (enumeration)
   Val_Cmd : SINT; {access Read Only}   // Device Command 0=None, 1=Stop, 2=Start
   Val_Fdbk : SINT; {access Read Only}   // Device Feedback 0=Stopped, 1=Running
   Val_Sts : SINT; {access Read Only}   // Device Confirmed Sts 0=? 1=Stopped, 2=Running, 7=Stopping, 8=Starting, 33=Disabled
   Val_Fault : SINT; {access Read Only}   // Device Fault Status 0=None, 16=Fail to Start, 17 = Fail to Stop, 32=I/O Fault, 34=Config Error
   Val_Mode : ALIAS FOR Mode.Val; {access Read Only}
   Val_Owner : DINT; {access Read Only}   // Current Object Owner ID (0=not owned)
   Val_Notify : SINT; {access Read Only}   // Current Alarm Level and Acknowledgement (enumeration)
   Sts_Stopped : BOOL := 1; {access Read Only, visible}   // 1=Motor requested to stop and is confirmed stopped
   Sts_Starting : BOOL; {access Read Only, visible}   // 1=Motor requested to run and awaiting run feedback
   Sts_Running : BOOL; {access Read Only, visible}   // 1=Motor requested to run and is confirmed running
   Sts_Stopping : BOOL; {access Read Only, visible}   // 1=Motor requested to stop and awaiting stopped feedback
   Sts_Available : BOOL; {access Read Only}   // 1=Motor available for control by automation (Prog)
   Sts_Bypass : BOOL; {access Read Only}   // 1=Bypassable Interlocks and Permissives are Bypassed
   Sts_BypActive : BOOL; {access Read Only}   // 1=Bypassing Active (Bypassed or Maintenance)
   Sts_Disabled : BOOL; {access Read Only}   // 1=Motor is Disabled
   Sts_NotRdy : BOOL; {access Read Only}   // 1=Device Not Ready, see detail bits for reason
   Nrdy_Disabled : BOOL; {access Read Only}   // 1=Device Not Ready: Device Disabled by Maintenance
   Nrdy_CfgErr : BOOL; {access Read Only}   // 1=Device Not Ready: Configuration Error
   Nrdy_Intlk : BOOL; {access Read Only}   // 1=Device Not Ready: Interlock Not OK
   Nrdy_Perm : BOOL; {access Read Only}   // 1=Device Not Ready: Permissive Not OK
   Nrdy_OperPrio : BOOL; {access Read Only}   // 1=Device Not Ready: Operator State 0 Priority Command Requires Reset
   Nrdy_Fail : BOOL; {access Read Only}   // 1=Device Not Ready: Device Failure (Shed Requires Reset)
   Nrdy_IOFault : BOOL; {access Read Only}   // 1=Device Not Ready: I/O Fault (Shed Requires Reset)
   Nrdy_NoMode : BOOL; {access Read Only}   // 1=Device Not Ready: Device Logic Disabled / NO Mode
   Sts_MaintByp : BOOL; {access Read Only}   // 1=A Maintenance Bypass is Active, display icon
   Sts_AlmInh : BOOL; {access Read Only}   // 1=An Alarm is Shelved, Disabled or Suppressed: display icon
   Sts_Err : BOOL; {access Read Only, visible}   // 1=Error in Config: see detail bits for reason
   Err_Timer : BOOL; {access Read Only}   // 1=Error in Config: Start/Stop Check timer preset (use 0 to 2147483)
   Err_Sim : BOOL; {access Read Only}   // 1=Error in Config: Simulation timer preset (use 0 to 2147483)
   Err_Alarm : BOOL; {access Read Only}   // 1=Error in Config: Alarm Min On Time, Shelf Time, Severity
   Sts_Hand : ALIAS FOR Mode.Sts_Hand; {access Read Only, visible}
   Sts_Maint : ALIAS FOR Mode.Sts_Maint; {access Read Only, visible}
   Sts_Ovrd : ALIAS FOR Mode.Sts_Ovrd; {access Read Only, visible}
   Sts_Prog : ALIAS FOR Mode.Sts_Prog; {access Read Only, visible}
   Sts_Oper : ALIAS FOR Mode.Sts_Oper; {access Read Only, visible}
   Sts_ProgOperLock : ALIAS FOR Mode.Sts_ProgOperLock; {access Read Only}
   Sts_NoMode : ALIAS FOR Mode.Sts_NoMode; {access Read Only}
   Sts_MAcqRcvd : ALIAS FOR Mode.Sts_MAcqRcvd; {access Read Only}
   Sts_FailToStart : ALIAS FOR FailToStart.Inp;   // 1=Motor Failed to Start (one-shot)
   Alm_FailToStart : ALIAS FOR FailToStart.Alm;   // 1=Motor Fail to Start Alarm
   Ack_FailToStart : ALIAS FOR FailToStart.Ack;   // 1=Fail to Start Alarm has been acknowledged
   Sts_FailToStartDisabled : ALIAS FOR FailToStart.Disabled;   // 1=Fail to Start Alarm has been Disabled by Maintenance
   Sts_FailToStartShelved : ALIAS FOR FailToStart.Shelved;   // 1=Fail to Start Alarm has been Shelved by Operator
   Sts_FailToStartSuppressed : ALIAS FOR FailToStart.Suppressed;   // 1=Fail to Start Alarm has been Suppressed by Program
   Sts_FailToStop : ALIAS FOR FailToStop.Inp;   // 1=Motor Failed to Stop
   Alm_FailToStop : ALIAS FOR FailToStop.Alm;   // 1=Motor Fail to Stop Alarm
   Ack_FailToStop : ALIAS FOR FailToStop.Ack;   // 1=Fail to Stop Alarm has been acknowledged
   Sts_FailToStopDisabled : ALIAS FOR FailToStop.Disabled;   // 1=Fail to Stop Alarm has been Disabled by Maintenance
   Sts_FailToStopShelved : ALIAS FOR FailToStop.Shelved;   // 1=Fail to Stop Alarm has been Shelved by Operator
   Sts_FailToStopSuppressed : ALIAS FOR FailToStop.Suppressed;   // 1=Fail to Stop Alarm has been Suppressed by Program
   Sts_IntlkTrip : ALIAS FOR IntlkTrip.Inp;   // 1=Motor stopped by an Interlock NOT OK (one-shot)
   Alm_IntlkTrip : ALIAS FOR IntlkTrip.Alm;   // 1=Alarm: Motor stopped by an Interlock NOT OK
   Ack_IntlkTrip : ALIAS FOR IntlkTrip.Ack;   // 1=Interlock Trip Alarm has been acknowledged
   Sts_IntlkTripDisabled : ALIAS FOR IntlkTrip.Disabled;   // 1=Interlock Trip Alarm has been Disabled by Maintenance
   Sts_IntlkTripShelved : ALIAS FOR IntlkTrip.Shelved;   // 1=Interlock Trip Alarm has been Shelved by Operator
   Sts_IntlkTripSuppressed : ALIAS FOR IntlkTrip.Suppressed;   // 1=Interlock Trip Alarm has been Suppressed by Program
   Sts_IOFault : ALIAS FOR IOFault.Inp;   // I/O Comm Fault Status (0=OK, 1=Bad)
   Alm_IOFault : ALIAS FOR IOFault.Alm;   // 1=I/O Fault Alarm
   Ack_IOFault : ALIAS FOR IOFault.Ack;   // 1=I/O Fault Alarm has been acknowledged
   Sts_IOFaultDisabled : ALIAS FOR IOFault.Disabled;   // 1=I/O Fault Alarm has been Disabled by Maintenance
   Sts_IOFaultShelved : ALIAS FOR IOFault.Shelved;   // 1=I/O Fault Alarm has been Shelved by Operator
   Sts_IOFaultSuppressed : ALIAS FOR IOFault.Suppressed;   // 1=I/O Fault Alarm has been Suppressed by Program
   Rdy_Start : BOOL; {access Read Only}   // 1=Ready to receive OCmd_Start (enables HMI button)
   Rdy_Stop : BOOL; {access Read Only}   // 1=Ready to receive OCmd_Stop (enables HMI button)
   Rdy_Bypass : BOOL; {access Read Only}   // 1=Ready to receive OCmd_Bypass (enables HMI button)
   Rdy_Check : BOOL; {access Read Only}   // 1=Ready to receive OCmd_Check (enables HMI button)
   Rdy_Disable : BOOL; {access Read Only}   // 1=Ready to receive MCmd_Disable (enables HMI button)
   Rdy_Enable : BOOL; {access Read Only}   // 1=Ready to receive MCmd_Enable (enables HMI button)
   Rdy_Reset : BOOL; {access Read Only}   // 1=At least one Alarm or Latched Shed requires Reset
   Rdy_ResetAckAll : BOOL; {access Read Only}   // 1=At least one Alarm or latched Shed condition requires Reset or Ack
   P_Motor : BOOL;   // Unique Parameter Name for auto - discovery
END_VAR
VAR
   Mode : P_Mode := (Cfg_PCmdClear := 1, Cfg_OvrdOverLock := 1, Sts_Oper := 1, Rdy_OAcq := 1);   // Motor Mode Selection
   IOFault : P_Alarm := (Cfg_AckReqd := 1, Cfg_AllowShelve := 1, Cfg_AllowDisable := 1, Cfg_PCmdClear := 1, Cfg_Severity := 1000, Cfg_AlmMinOnT := 5, PCfg_AllowExist := 1, Ack := 1);   // I/O Fault Alarm
   IntlkTrip : P_Alarm := (Cfg_AckReqd := 1, Cfg_AllowShelve := 1, Cfg_AllowDisable := 1, Cfg_PCmdClear := 1, Cfg_Severity := 500, Cfg_AlmMinOnT := 5, PCfg_AllowExist := 1, Ack := 1);   // Interlock Trip Alarm
   FailToStop : P_Alarm := (Cfg_AckReqd := 1, Cfg_AllowShelve := 1, Cfg_AllowDisable := 1, Cfg_PCmdClear := 1, Cfg_Severity := 1000, Cfg_AlmMinOnT := 5, PCfg_AllowExist := 1, Ack := 1);   // Motor Failed to Stop Alarm
   FailToStart : P_Alarm := (Cfg_AckReqd := 1, Cfg_AllowShelve := 1, Cfg_AllowDisable := 1, Cfg_PCmdClear := 1, Cfg_Severity := 1000, Cfg_AlmMinOnT := 5, PCfg_AllowExist := 1, Ack := 1);   // Motor Failed to Start Alarm
   Cfg_Tag : STRING_20 := 'P_Motor';   // Tagname for display on HMI
   Cfg_Label : STRING_20 := 'Motor Control';   // Label for graphic symbol displayed on HMI
   Cfg_Desc : STRING_40 := 'Single Speed Motor';   // Description for display on HMI
   Wrk_Run : BOOL; {access None}   // 1=Motor should be "running", 0=should be "stopped"
   Wrk_SimRunT : TIMER; {access None}   // Simulation Delay until Running
   Wrk_StopT : TIMER; {access Read Only}   // Stop Check Timer
   Wrk_StartT : TIMER; {access Read Only}   // Start Check Timer
   Wrk_SimStopT : TIMER; {access None}   // Simulation Delay until Stopped
   Wrk_RunFdbk : BOOL; {access None}   // Run Feedback based on mode, simulation, etc. 1=running
   Wrk_Notify : DINT; {access None}   // Buffer for building Val_Notify
   Wrk_Bypass : BOOL; {access None}   // Internal Bypassable Permissives and Interlocks are Bypassed flag
   Wrk_Disabled : BOOL; {access None}   // Internal Motor is Disabled
   Inf_Tab : SINT;   // Tab to display (FTView ME)
   Wrk_Cmd : SINT; {access None}   // Buffer for building Val_Cmd
   Wrk_Sts : SINT; {access None}   // Buffer for building Val_Sts
   Wrk_Fault : SINT; {access None}   // Buffer for building Val_Fault
   Wrk_Retrigger : BOOL; {access None}   // Maint Start issued while running or Stop while stopped
   Inf_Type : STRING_16 := 'P_Motor'; {access Read Only}   // Type identifier for HMI navigation
   Inf_Lib : STRING_12 := 'RA-BAS'; {access Read Only}   // Display Library for Faceplate call-up
   Wrk_SrcQ : SINT; {access None}   // Register for building Source / Quality enumeration
   Wrk_NotRdyONS : BOOL; {access None}   // Assert Stop on One-Shot of Sts_NotRdy
   Wrk_NotRdy : BOOL; {access None}   // Device Not Ready conditions excluding shed latches
   Wrk_StopInhT : TIMER; {access None}   // Local Stop Inhibit Timer
   Wrk_StartInhT : TIMER; {access None}   // Local Start Inhibit Timer
   Wrk_NoLongerSim : BOOL; {access None}   // Switched from Simulated to Real Motor this scan
END_VAR

ROUTINE EnableInFalse   (* ladder *)
// Disabled is asserted; Outputs OFF; Run Status shown but Alarms disabled
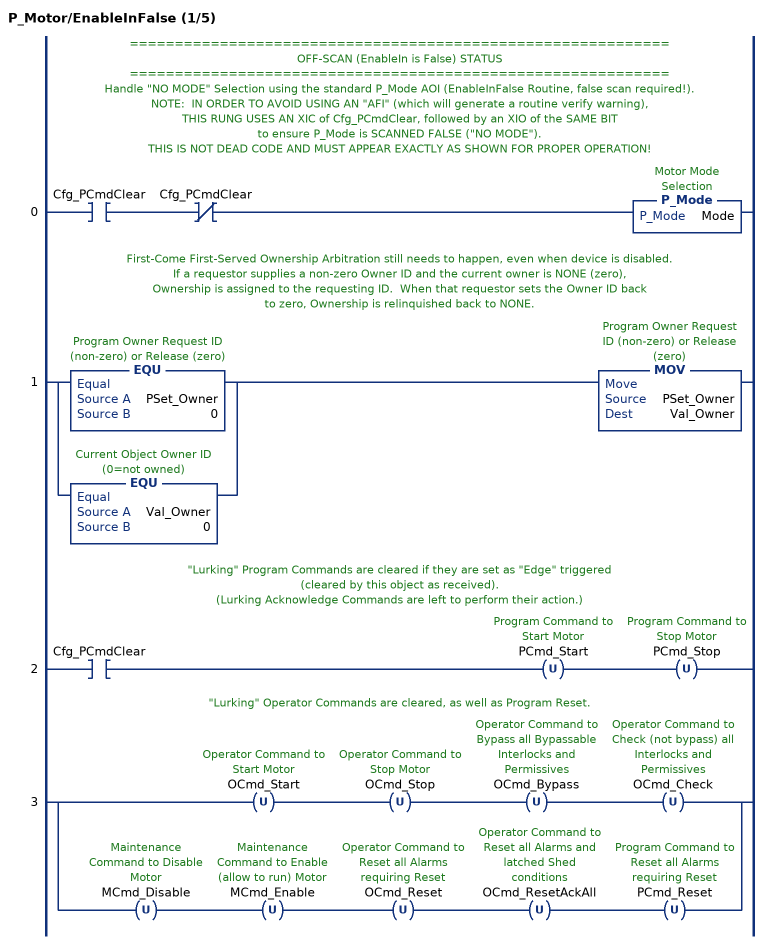
   // ============================================================
   // OFF-SCAN (EnableIn is False) STATUS
   // ============================================================
   // Handle "NO MODE" Selection using the standard P_Mode AOI (EnableInFalse Routine, false scan required!).
   // NOTE:  IN ORDER TO AVOID USING AN "AFI" (which will generate a routine verify warning),
   // THIS RUNG USES AN XIC of Cfg_PCmdClear, followed by an XIO of the SAME BIT
   // to ensure P_Mode is SCANNED FALSE ("NO MODE").
   // THIS IS NOT DEAD CODE AND MUST APPEAR EXACTLY AS SHOWN FOR PROPER OPERATION!
   0: XIC(Cfg_PCmdClear)XIO(Cfg_PCmdClear)P_Mode(Mode);
   // First-Come First-Served Ownership Arbitration still needs to happen, even when device is disabled.
   // If a requestor supplies a non-zero Owner ID and the current owner is NONE (zero),
   // Ownership is assigned to the requesting ID.  When that requestor sets the Owner ID back
   // to zero, Ownership is relinquished back to NONE.
   1: [EQU(PSet_Owner,0) ,EQU(Val_Owner,0) ]MOV(PSet_Owner,Val_Owner);
   // "Lurking" Program Commands are cleared if they are set as "Edge" triggered
   // (cleared by this object as received).
   // (Lurking Acknowledge Commands are left to perform their action.)
   2: XIC(Cfg_PCmdClear)OTU(PCmd_Start)OTU(PCmd_Stop);
   // "Lurking" Operator Commands are cleared, as well as Program Reset.
   3: [OTU(OCmd_Start) OTU(OCmd_Stop) OTU(OCmd_Bypass) OTU(OCmd_Check) ,OTU(MCmd_Disable) OTU(MCmd_Enable) OTU(OCmd_Reset) OTU(OCmd_ResetAckAll) OTU(PCmd_Reset) ];
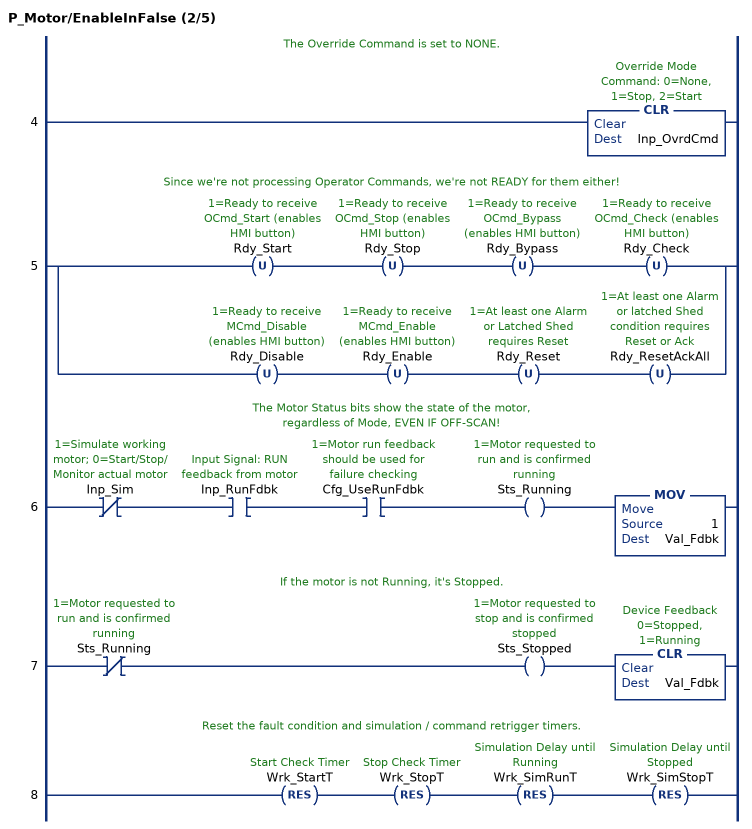
   // The Override Command is set to NONE.
   4: CLR(Inp_OvrdCmd);
   // Since we're not processing Operator Commands, we're not READY for them either!
   5: [OTU(Rdy_Start) OTU(Rdy_Stop) OTU(Rdy_Bypass) OTU(Rdy_Check) ,OTU(Rdy_Disable) OTU(Rdy_Enable) OTU(Rdy_Reset) OTU(Rdy_ResetAckAll) ];
   // The Motor Status bits show the state of the motor,
   // regardless of Mode, EVEN IF OFF-SCAN!
   6: XIO(Inp_Sim)XIC(Inp_RunFdbk)XIC(Cfg_UseRunFdbk)OTE(Sts_Running)MOV(1,Val_Fdbk);
   // If the motor is not Running, it's Stopped.
   7: XIO(Sts_Running)OTE(Sts_Stopped)CLR(Val_Fdbk);
   // Reset the fault condition and simulation / command retrigger timers.
   8: RES(Wrk_StartT)RES(Wrk_StopT)RES(Wrk_SimRunT)RES(Wrk_SimStopT);
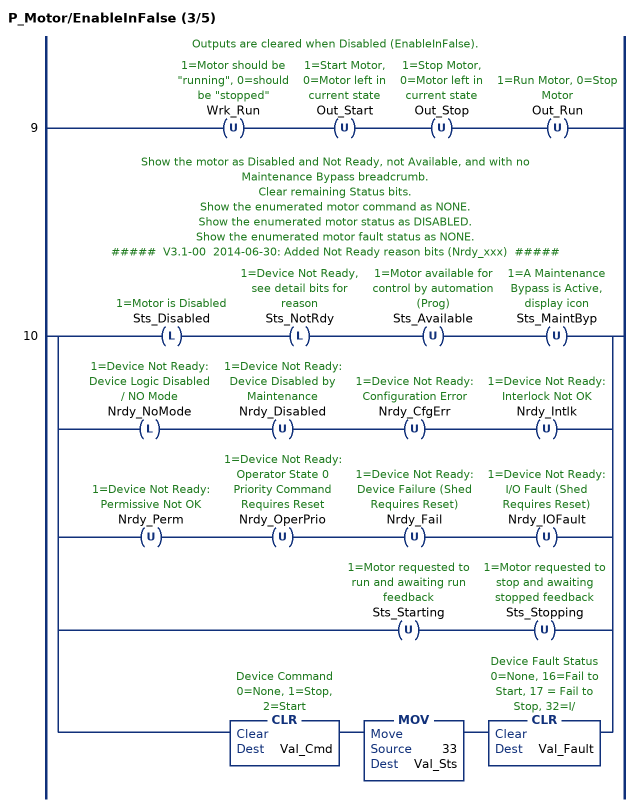
   // Outputs are cleared when Disabled (EnableInFalse).
   9: OTU(Wrk_Run)OTU(Out_Start)OTU(Out_Stop)OTU(Out_Run);
   // Show the motor as Disabled and Not Ready, not Available, and with no
   // Maintenance Bypass breadcrumb.
   // Clear remaining Status bits.
   // Show the enumerated motor command as NONE.
   // Show the enumerated motor status as DISABLED.
   // Show the enumerated motor fault status as NONE.
   // #####  V3.1-00  2014-06-30: Added Not Ready reason bits (Nrdy_xxx)  #####
   10: [OTL(Sts_Disabled) OTL(Sts_NotRdy) OTU(Sts_Available) OTU(Sts_MaintByp) ,OTL(Nrdy_NoMode) OTU(Nrdy_Disabled) OTU(Nrdy_CfgErr) OTU(Nrdy_Intlk) ,OTU(Nrdy_Perm) OTU(Nrdy_OperPrio) OTU(Nrdy_Fail) OTU(Nrdy_IOFault) ,OTU(Sts_Starting) OTU(Sts_Stopping) ,CLR(Val_Cmd) MOV(33,Val_Sts) CLR(Val_Fault) ];
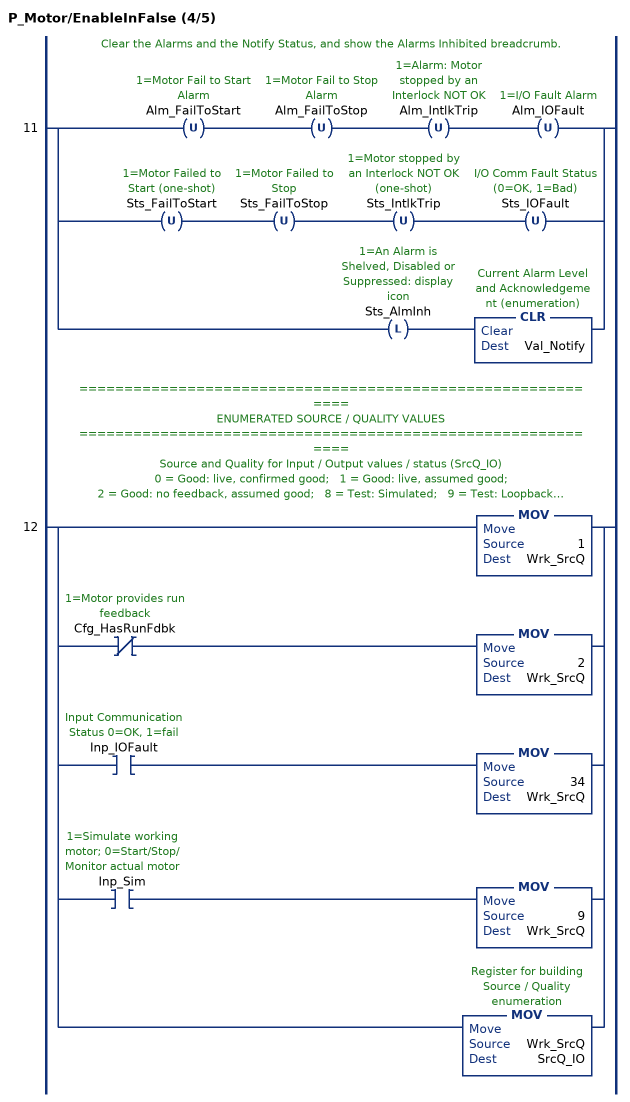
   // Clear the Alarms and the Notify Status, and show the Alarms Inhibited breadcrumb.
   11: [OTU(Alm_FailToStart) OTU(Alm_FailToStop) OTU(Alm_IntlkTrip) OTU(Alm_IOFault) ,OTU(Sts_FailToStart) OTU(Sts_FailToStop) OTU(Sts_IntlkTrip) OTU(Sts_IOFault) ,OTL(Sts_AlmInh) CLR(Val_Notify) ];
   // ============================================================
   // ENUMERATED SOURCE / QUALITY VALUES
   // ============================================================
   // Source and Quality for Input / Output values / status (SrcQ_IO)
   // 0 = Good: live, confirmed good;   1 = Good: live, assumed good;
   // 2 = Good: no feedback, assumed good;   8 = Test: Simulated;   9 = Test: Loopback;
   // 10 = Test: Manually Entered;   16 = Uncertain: Live, off-spec;
   // 17 = Uncertain, Substituted at Device / Bus;   18 = Uncertain, Substituted at AOI;
   // 19 = Uncertain, using last known good;    20 = Uncertain, using replacement value;
   // 32 = Bad, Signal Failure;   33 = Bad, Channel Fault;
   // 34 = Bad, Module / Comms Fault;   35 = Bad, Invalid Configuration
   // #####  V3.1-00  2014-06-30:  Added rung for Source/Quality enumerations.  #####
   12: [MOV(1,Wrk_SrcQ) ,XIO(Cfg_HasRunFdbk) MOV(2,Wrk_SrcQ) ,XIC(Inp_IOFault) MOV(34,Wrk_SrcQ) ,XIC(Inp_Sim) MOV(9,Wrk_SrcQ) ,MOV(Wrk_SrcQ,SrcQ_IO) ];
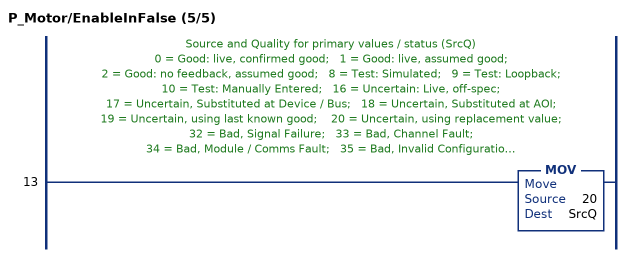
   // Source and Quality for primary values / status (SrcQ)
   // 0 = Good: live, confirmed good;   1 = Good: live, assumed good;
   // 2 = Good: no feedback, assumed good;   8 = Test: Simulated;   9 = Test: Loopback;
   // 10 = Test: Manually Entered;   16 = Uncertain: Live, off-spec;
   // 17 = Uncertain, Substituted at Device / Bus;   18 = Uncertain, Substituted at AOI;
   // 19 = Uncertain, using last known good;    20 = Uncertain, using replacement value;
   // 32 = Bad, Signal Failure;   33 = Bad, Channel Fault;
   // 34 = Bad, Module / Comms Fault;   35 = Bad, Invalid Configuration
   // #####  V3.1-00  2014-06-30:  Added rung for Source/Quality enumerations.  #####
   13: MOV(20,SrcQ);
END_ROUTINE

ROUTINE Logic   (* ladder *)
// Normal Scan: control / monitor single speed motor
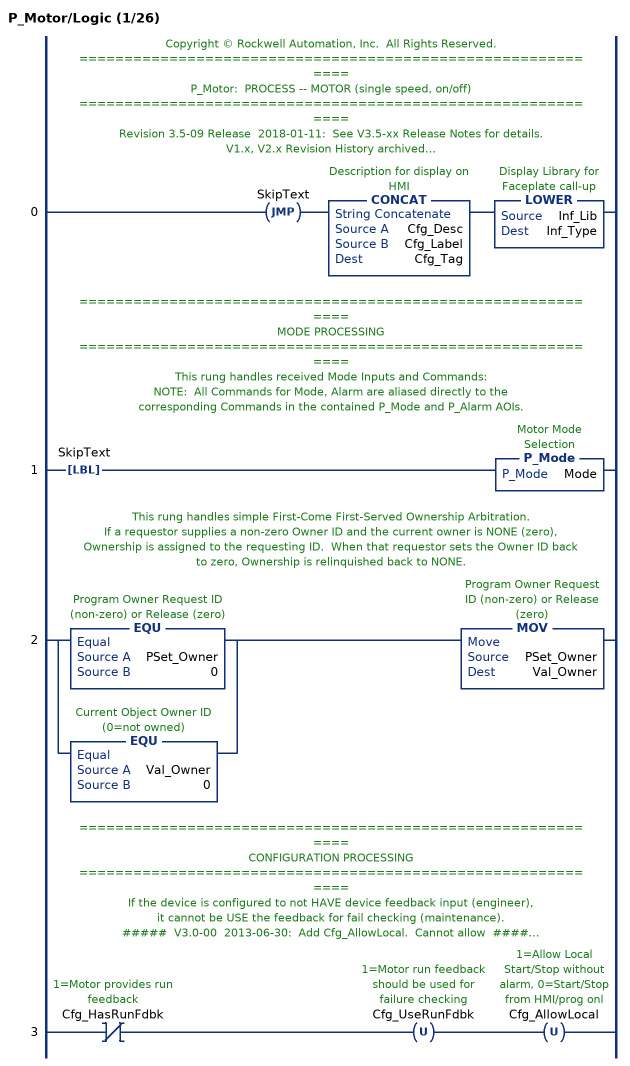
   // Copyright © Rockwell Automation, Inc.  All Rights Reserved.
   // ============================================================
   // P_Motor:  PROCESS -- MOTOR (single speed, on/off)
   // ============================================================
   // Revision 3.5-09 Release  2018-01-11:  See V3.5-xx Release Notes for details.
   // V1.x, V2.x Revision History archived.
   // V3.0-00  2013-06-30:  Added Inf_Lib.  Added Cfg_AllowLocal, Cfg_OperStopPrio,
   // Cfg_HasOvldObj.  Using P_Alarm V3.0, P_Mode V3.0.
   // V3.0-01  2013-07-30:  Modified Parameter descriptions only.
   // V3.0-02  2013-09-03:  Modified to ensure Out_Stop always pulses
   // whenever a stop command is received, regardless of run
   // feedback state.  Modified Parameter descriptions.
   // V3.0-03  2013-09-10:  Corrected modification above for operation
   // in simulation and for all start, stop and not-ready conditions.
   // V3.0-04  2013-10-30:  Corrected Parameter descriptions and default
   // configuration values for alarms only.
   // Modified default Parameter values.
   // V3.0-05  2014-06-12:  Modified Out_Stop action on shed,
   // allow Operator retrigger of Stop command.
   // V3.1-00  2014-07-08:  Modified to use P_Alarm, P_Mode V3.1. Added
   // Not Ready reason bits (Nrdy_Xxxxx), source/quality values
   // (SrcQ). Modified to consistently use alias tag names.
   // V3.1-01  2014-09-03:  Resolved held "Stopping" status. Exposed fail timers
   // ACC/PRE (read-only). Corrections to Nrdy_ trip and
   // reset logic. Using P_Alarm, P_Mode V3.1-01.
   // V3.1-02  2014-09-30:  Unchanged, but using P_Alarm V3.1-02.
   // V3.1-03  2015-01-16;  Modified stop retriggering to handle asynchronous Prog mode owner.
   // V3.1-04 Patch01  2015-09-25: Modified handling of run feedback latch on prescan.
   // Modified to correct issue with loss of run feedback.
   // V3.5-01  2016-01-29: Unchanged, but using P_Alarm V3.5-01.
   // V3.5-04  2016-09-30: Modified to align with actual device state on
   // transition from Sim to real motor.
   // V3.5-09  2018-01-11:  Modified to correct indication of motor RUNNING status in HAND
   // mode, regardless of interlock/stop conditions.
   // ============================================================
   // This Instruction controls and monitors a single-speed motor
   // (FVNR, soft-start, etc.) and provides:
   // *  Monitoring of run feedback, display of actual motor status
   // *  Detection of Failure to Start, Failure to Stop
   // *  Monitoring of a Permissive condition to allow starting
   // * Monitoring of an Interlock condition to stop / prevent starting
   // * Simulation, providing feedback of a working motor while disabling outputs
   // * Monitoring of I/O communication faults
   // * Alarms for Fail to Start, Fail to Stop, Interlock Trip, I/O Fault
   // * Options to shed (stop motor) on Fail to Start or I/O Fault
   // * Option to automatically reset faults and alarms when operator commands
   // motor to start or stop
   // * Supports HMI "breadcrumbs" for Alarm Inhibited, Bad Configuration,
   // Not Ready, Maintenance Bypass Active
   // * "Available" status for use by automation logic to know whether motor
   // can be controlled by other objects.
   // Modes are provided by a P_Mode AOI instance.
   // Alarms are provided by P_Alarm AOI instances.
   // Modes of operation: Operator, Program, Override, Maintenance, Hand
   // ============================================================
   // SHOW LOCAL STRINGS
   // ============================================================
   // The STRINGs containing the text associated with each instance of this
   // instruction cannot be Input or Output Parameters, because STRINGs are not
   //  'atomic' types. (Inputs and Outputs must be SINT, INT, DINT, REAL, or BOOL.)
   // In order to make it easier to find and configure these STRINGs, this rung
   // was added.  THE JMP (and the LBL on the following rung)
   // MUST NOT BE REMOVED!!!
   // To view the STRINGs, go to the instruction instance (in LD or FBD), RIGHT-click
   // to bring up the context menu and select "Open Instruction Logic".
   // This rung will appear with the STRING values for the selected instance.
   // You may double-click the STRING values here to modify them as well.
   0: JMP(SkipText)CONCAT(Cfg_Desc,Cfg_Label,Cfg_Tag)LOWER(Inf_Lib,Inf_Type);
   // ============================================================
   // MODE PROCESSING
   // ============================================================
   // This rung handles received Mode Inputs and Commands:
   // NOTE:  All Commands for Mode, Alarm are aliased directly to the
   // corresponding Commands in the contained P_Mode and P_Alarm AOIs.
   1: LBL(SkipText)P_Mode(Mode);
   // This rung handles simple First-Come First-Served Ownership Arbitration.
   // If a requestor supplies a non-zero Owner ID and the current owner is NONE (zero),
   // Ownership is assigned to the requesting ID.  When that requestor sets the Owner ID back
   // to zero, Ownership is relinquished back to NONE.
   2: [EQU(PSet_Owner,0) ,EQU(Val_Owner,0) ]MOV(PSet_Owner,Val_Owner);
   // ============================================================
   // CONFIGURATION PROCESSING
   // ============================================================
   // If the device is configured to not HAVE device feedback input (engineer),
   // it cannot be USE the feedback for fail checking (maintenance).
   // #####  V3.0-00  2013-06-30:  Add Cfg_AllowLocal.  Cannot allow  #####
   // #####  local start/stop  if run feedback does not exist to monitor for it.  #####
   3: XIO(Cfg_HasRunFdbk)OTU(Cfg_UseRunFdbk)OTU(Cfg_AllowLocal);
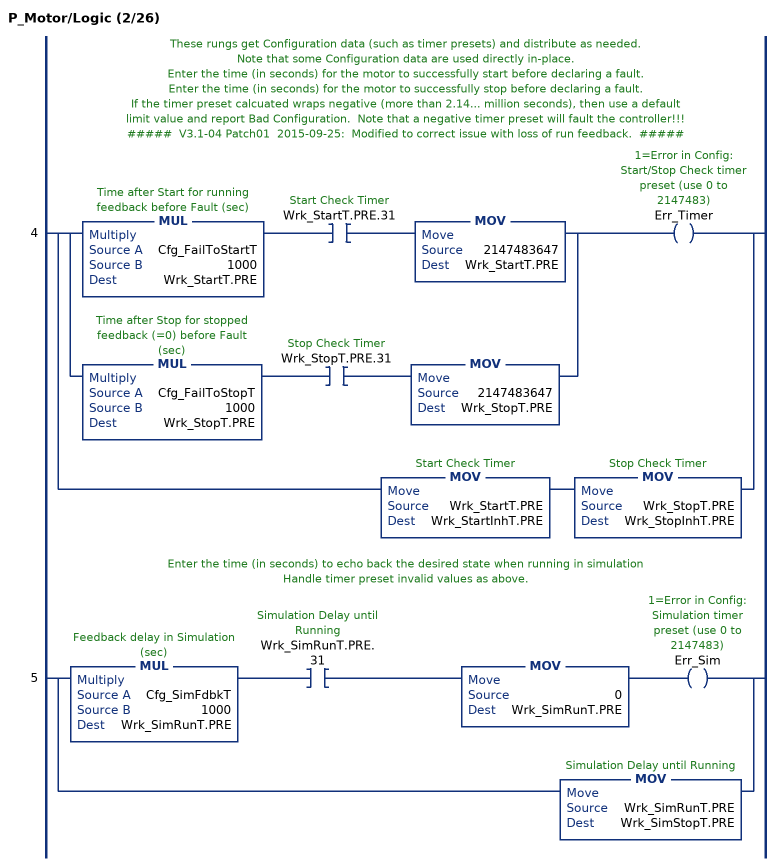
   // These rungs get Configuration data (such as timer presets) and distribute as needed.
   // Note that some Configuration data are used directly in-place.
   // Enter the time (in seconds) for the motor to successfully start before declaring a fault.
   // Enter the time (in seconds) for the motor to successfully stop before declaring a fault.
   // If the timer preset calcuated wraps negative (more than 2.14... million seconds), then use a default
   // limit value and report Bad Configuration.  Note that a negative timer preset will fault the controller!!!
   // #####  V3.1-04 Patch01  2015-09-25:  Modified to correct issue with loss of run feedback.  #####
   4: [[MUL(Cfg_FailToStartT,1000,Wrk_StartT.PRE) XIC(Wrk_StartT.PRE.31) MOV(2147483647,Wrk_StartT.PRE) ,MUL(Cfg_FailToStopT,1000,Wrk_StopT.PRE) XIC(Wrk_StopT.PRE.31) MOV(2147483647,Wrk_StopT.PRE) ] OTE(Err_Timer) ,MOV(Wrk_StartT.PRE,Wrk_StartInhT.PRE) MOV(Wrk_StopT.PRE,Wrk_StopInhT.PRE) ];
   // Enter the time (in seconds) to echo back the desired state when running in simulation
   // Handle timer preset invalid values as above.
   5: [MUL(Cfg_SimFdbkT,1000,Wrk_SimRunT.PRE) XIC(Wrk_SimRunT.PRE.31) MOV(0,Wrk_SimRunT.PRE) OTE(Err_Sim) ,MOV(Wrk_SimRunT.PRE,Wrk_SimStopT.PRE) ];
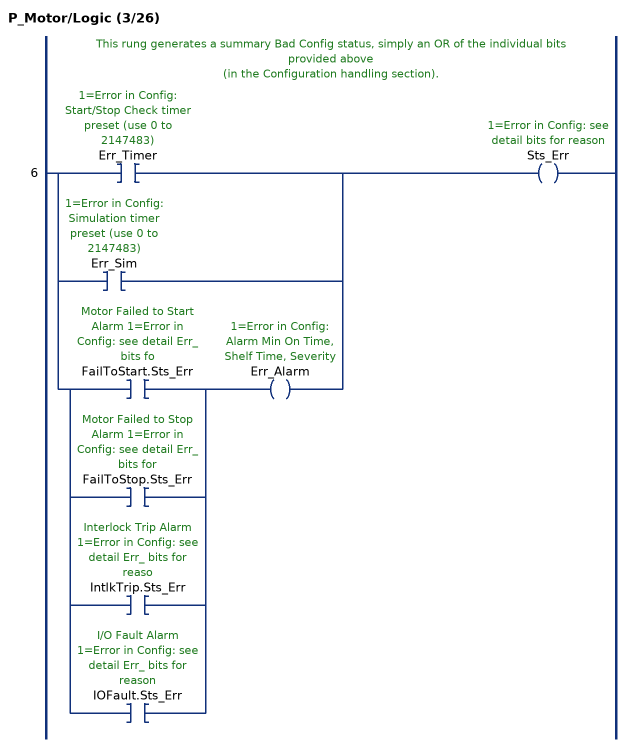
   // This rung generates a summary Bad Config status, simply an OR of the individual bits provided above
   // (in the Configuration handling section).
   6: [XIC(Err_Timer) ,XIC(Err_Sim) ,[XIC(FailToStart.Sts_Err) ,XIC(FailToStop.Sts_Err) ,XIC(IntlkTrip.Sts_Err) ,XIC(IOFault.Sts_Err) ] OTE(Err_Alarm) ]OTE(Sts_Err);
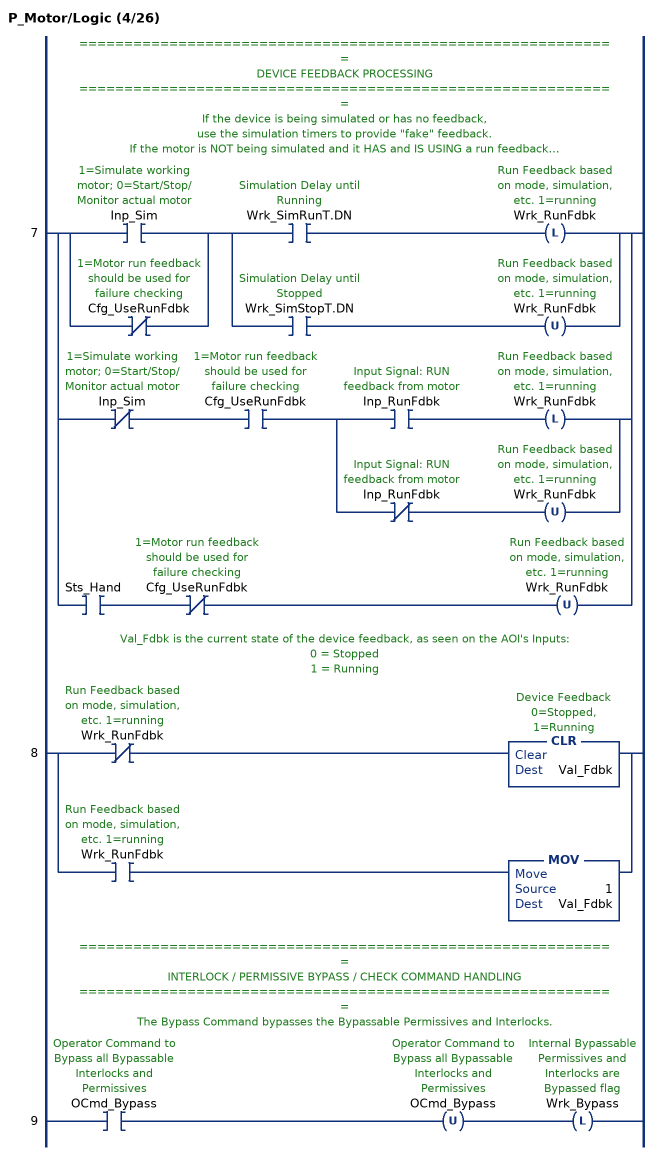
   // ============================================================
   // DEVICE FEEDBACK PROCESSING
   // ============================================================
   // If the device is being simulated or has no feedback,
   // use the simulation timers to provide "fake" feedback.
   // If the motor is NOT being simulated and it HAS and IS USING a run feedback,
   // use the state of the run feedback input as the motor run state.
   7: [[XIC(Inp_Sim) ,XIO(Cfg_UseRunFdbk) ] [XIC(Wrk_SimRunT.DN) OTL(Wrk_RunFdbk) ,XIC(Wrk_SimStopT.DN) OTU(Wrk_RunFdbk) ] ,XIO(Inp_Sim) XIC(Cfg_UseRunFdbk) [XIC(Inp_RunFdbk) OTL(Wrk_RunFdbk) ,XIO(Inp_RunFdbk) OTU(Wrk_RunFdbk) ] ,XIC(Sts_Hand) XIO(Cfg_UseRunFdbk) OTU(Wrk_RunFdbk) ];
   // Val_Fdbk is the current state of the device feedback, as seen on the AOI's Inputs:
   // 0 = Stopped
   // 1 = Running
   8: [XIO(Wrk_RunFdbk) CLR(Val_Fdbk) ,XIC(Wrk_RunFdbk) MOV(1,Val_Fdbk) ];
   // ============================================================
   // INTERLOCK / PERMISSIVE BYPASS / CHECK COMMAND HANDLING
   // ============================================================
   // The Bypass Command bypasses the Bypassable Permissives and Interlocks.
   9: XIC(OCmd_Bypass)OTU(OCmd_Bypass)OTL(Wrk_Bypass);
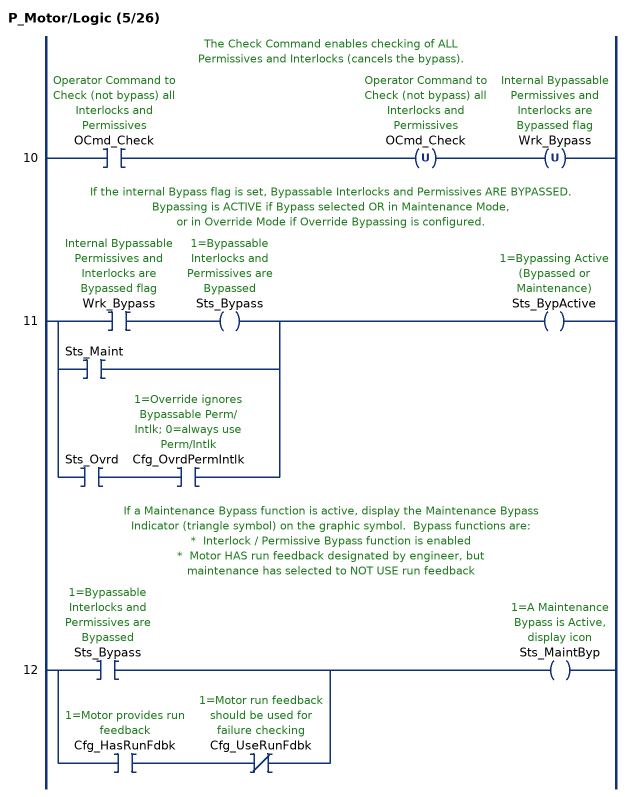
   // The Check Command enables checking of ALL
   // Permissives and Interlocks (cancels the bypass).
   10: XIC(OCmd_Check)OTU(OCmd_Check)OTU(Wrk_Bypass);
   // If the internal Bypass flag is set, Bypassable Interlocks and Permissives ARE BYPASSED.
   // Bypassing is ACTIVE if Bypass selected OR in Maintenance Mode,
   // or in Override Mode if Override Bypassing is configured.
   11: [XIC(Wrk_Bypass) OTE(Sts_Bypass) ,XIC(Sts_Maint) ,XIC(Sts_Ovrd) XIC(Cfg_OvrdPermIntlk) ]OTE(Sts_BypActive);
   // If a Maintenance Bypass function is active, display the Maintenance Bypass
   // Indicator (triangle symbol) on the graphic symbol.  Bypass functions are:
   // *  Interlock / Permissive Bypass function is enabled
   // *  Motor HAS run feedback designated by engineer, but
   // maintenance has selected to NOT USE run feedback
   12: [XIC(Sts_Bypass) ,XIC(Cfg_HasRunFdbk) XIO(Cfg_UseRunFdbk) ]OTE(Sts_MaintByp);
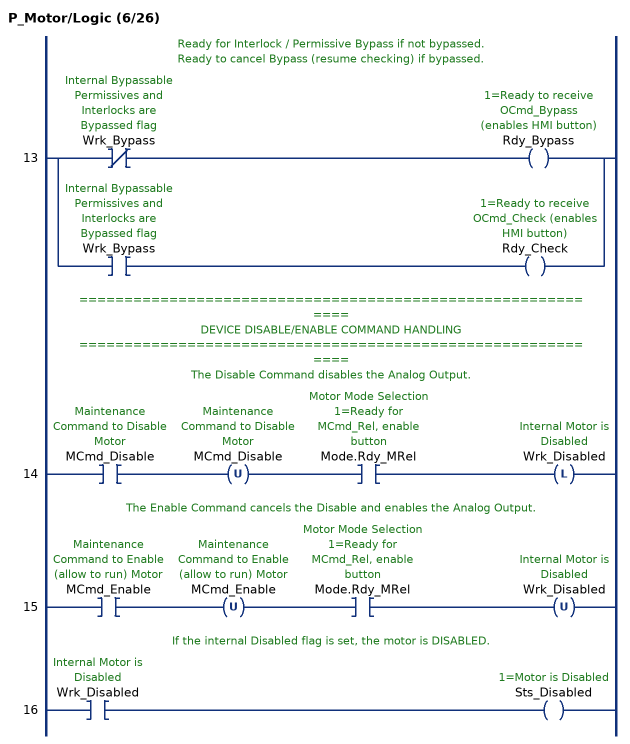
   // Ready for Interlock / Permissive Bypass if not bypassed.
   // Ready to cancel Bypass (resume checking) if bypassed.
   13: [XIO(Wrk_Bypass) OTE(Rdy_Bypass) ,XIC(Wrk_Bypass) OTE(Rdy_Check) ];
   // ============================================================
   // DEVICE DISABLE/ENABLE COMMAND HANDLING
   // ============================================================
   // The Disable Command disables the Analog Output.
   14: XIC(MCmd_Disable)OTU(MCmd_Disable)XIC(Mode.Rdy_MRel)OTL(Wrk_Disabled);
   // The Enable Command cancels the Disable and enables the Analog Output.
   15: XIC(MCmd_Enable)OTU(MCmd_Enable)XIC(Mode.Rdy_MRel)OTU(Wrk_Disabled);
   // If the internal Disabled flag is set, the motor is DISABLED.
   16: XIC(Wrk_Disabled)OTE(Sts_Disabled);
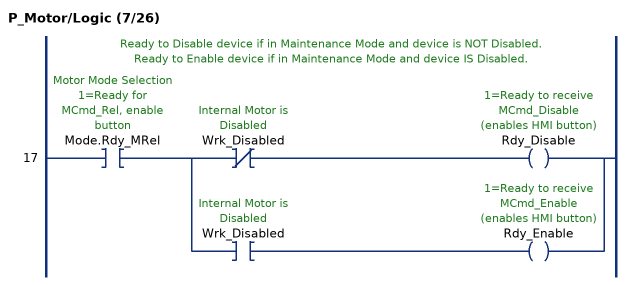
   // Ready to Disable device if in Maintenance Mode and device is NOT Disabled.
   // Ready to Enable device if in Maintenance Mode and device IS Disabled.
   17: XIC(Mode.Rdy_MRel)[XIO(Wrk_Disabled) OTE(Rdy_Disable) ,XIC(Wrk_Disabled) OTE(Rdy_Enable) ];
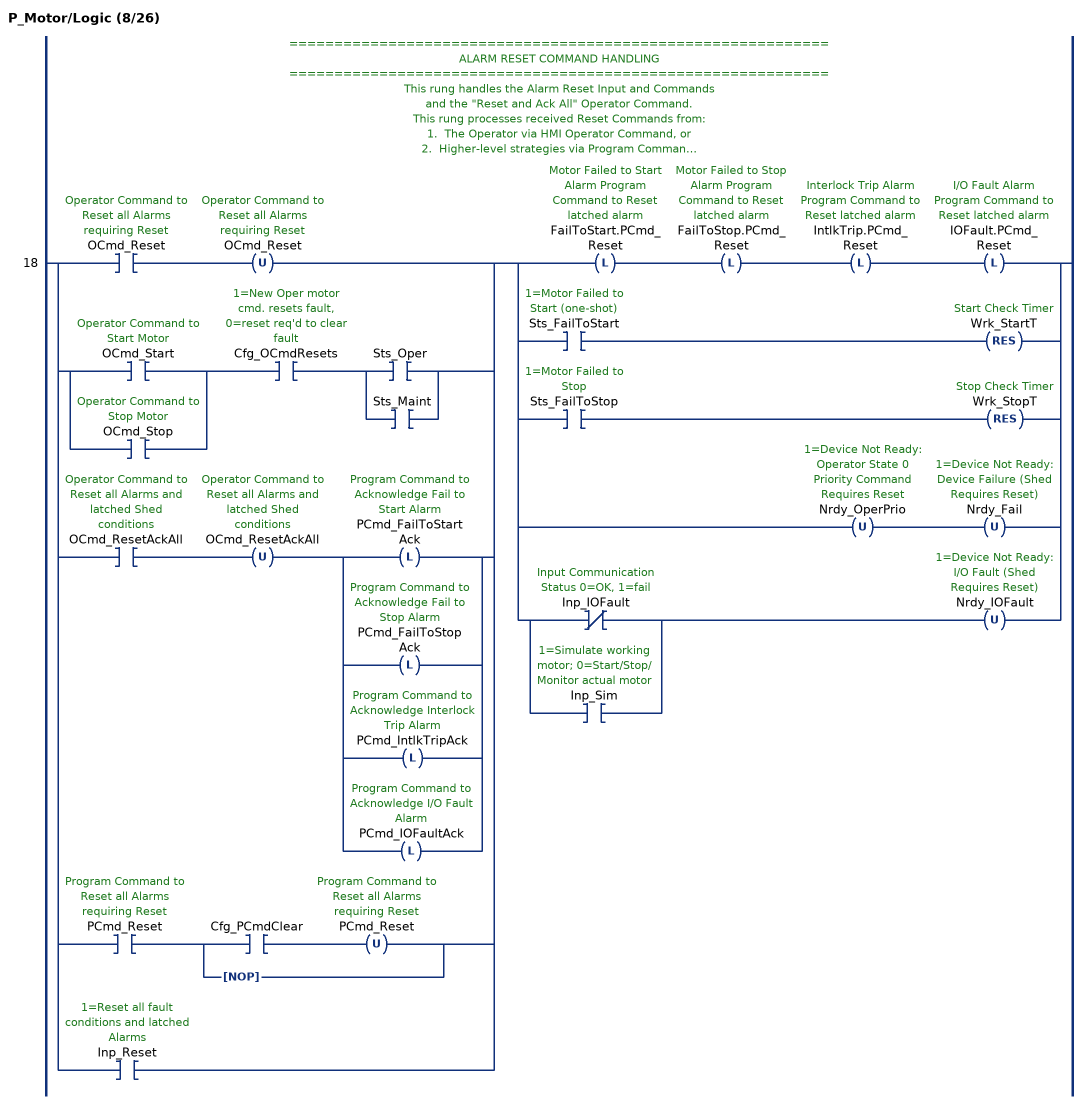
   // ============================================================
   // ALARM RESET COMMAND HANDLING
   // ============================================================
   // This rung handles the Alarm Reset Input and Commands
   // and the "Reset and Ack All" Operator Command.
   // This rung processes received Reset Commands from:
   // 1.  The Operator via HMI Operator Command, or
   // 2.  Higher-level strategies via Program Command
   // 3.  Pushbuttons or other block via Input
   // 4.  Resets initiated by other device Operator Commands (if configured to do so)
   // and forwards the Reset to ALL Alarms and latched Shed conditions.
   // #####  V3.1-00  2014-06-30: Added Not Ready reason bits (Nrdy_xxx)  #####
   // #####  V3.1-01  2014-08-29:  Corrections to Nrdy_ trip and reset logic.  #####
   18: [XIC(OCmd_Reset) OTU(OCmd_Reset) ,[XIC(OCmd_Start) ,XIC(OCmd_Stop) ] XIC(Cfg_OCmdResets) [XIC(Sts_Oper) ,XIC(Sts_Maint) ] ,XIC(OCmd_ResetAckAll) OTU(OCmd_ResetAckAll) [OTL(PCmd_FailToStartAck) ,OTL(PCmd_FailToStopAck) ,OTL(PCmd_IntlkTripAck) ,OTL(PCmd_IOFaultAck) ] ,XIC(PCmd_Reset) [XIC(Cfg_PCmdClear) OTU(PCmd_Reset) ,NOP() ] ,XIC(Inp_Reset) ][OTL(FailToStart.PCmd_Reset) OTL(FailToStop.PCmd_Reset) OTL(IntlkTrip.PCmd_Reset) OTL(IOFault.PCmd_Reset) ,XIC(Sts_FailToStart) RES(Wrk_StartT) ,XIC(Sts_FailToStop) RES(Wrk_StopT) ,OTU(Nrdy_OperPrio) OTU(Nrdy_Fail) ,[XIO(Inp_IOFault) ,XIC(Inp_Sim) ] OTU(Nrdy_IOFault) ];
